LIN {X 0,Y 574.038,Z 321.65,A -85,B 0,C 180,E1 -2269.624,E2 -2269.624} C_VEL
LIN {X 0,Y 574.354,Z 297.27,A -85,B 0,C 180,E1 -2272.482,E2 -2272.482} C_VEL
LIN {X 0,Y 574.708,Z 273.214,A -85,B 0,C 180,E1 -2275.342,E2 -2275.342} C_VEL
LIN {X 0,Y 574.694,Z 268.348,A -85,B 0,C 180,E1 -2275.925,E2 -2275.925} C_VEL
LIN {X 0,Y 573.245,Z 261.708,A -85,B 0,C 180,E1 -2276.811,E2 -2276.811} C_VEL
LIN {X 0,Y 573.247,Z 261.7,A -85,B 0,C 180,E1 -2279.488,E2 -2279.488} C_VEL
LIN {X 0,Y 573.255,Z 261.706,A -85,B 0,C 180,E1 -2282.645,E2 -2282.645} C_VEL
LIN {X 0,Y 573.209,Z 261.705,A -85,B 0,C 180,E1 -2285.188,E2 -2285.188} C_VEL
LIN {X 0,Y 573.237,Z 261.701,A -85,B 0,C 180,E1 -2287.808,E2 -2287.808} C_VEL
LIN {X 0,Y 573.248,Z 261.707,A -85,B 0,C 180,E1 -2290.525,E2 -2290.525} C_VEL
LIN {X 0,Y 573.211,Z 261.703,A -85,B 0,C 180,E1 -2293.362,E2 -2293.362} C_VEL
LIN {X 0,Y 573.241,Z 261.707,A -85,B 0,C 180,E1 -2296.332,E2 -2296.332} C_VEL
LIN {X 0,Y 573.23,Z 261.707,A -85,B 0,C 180,E1 -2298.543,E2 -2298.543} C_VEL
LIN {X 0,Y 573.239,Z 261.699,A -85,B 0,C 180,E1 -2301.298,E2 -2301.298} C_VEL
LIN {X 0,Y 573.192,Z 261.711,A -85,B 0,C 180,E1 -2304.022,E2 -2304.022} C_VEL
LIN {X 0,Y 573.257,Z 261.702,A -85,B 0,C 180,E1 -2306.517,E2 -2306.517} C_VEL
LIN {X 0,Y 573.23,Z 261.7,A -85,B 0,C 180,E1 -2309.119,E2 -2309.119} C_VEL
LIN {X 0,Y 573.228,Z 261.7,A -85,B 0,C 180,E1 -2311.435,E2 -2311.435} C_VEL
LIN {X 0,Y 573.243,Z 261.702,A -85,B 0,C 180,E1 -2314.589,E2 -2314.589} C_VEL
LIN {X 0,Y 573.235,Z 261.702,A -85,B 0,C 180,E1 -2317.662,E2 -2317.662} C_VEL
LIN {X 0,Y 573.271,Z 261.696,A -85,B 0,C 180,E1 -2320.67,E2 -2320.67} C_VEL
LIN {X 0,Y 573.241,Z 261.703,A -85,B 0,C 180,E1 -2323.622,E2 -2323.622} C_VEL
LIN {X 0,Y 573.276,Z 261.7,A -85,B 0,C 180,E1 -2325.807,E2 -2325.807} C_VEL
LIN {X 0,Y 573.269,Z 261.695,A -85,B 0,C 180,E1 -2328.745,E2 -2328.745} C_VEL
LIN {X 0,Y 573.253,Z 261.701,A -85,B 0,C 180,E1 -2331.54,E2 -2331.54} C_VEL
LIN {X 0,Y 573.271,Z 261.698,A -85,B 0,C 180,E1 -2334.372,E2 -2334.372} C_VEL
LIN {X 0,Y 573.304,Z 261.7,A -85,B 0,C 180,E1 -2337.892,E2 -2337.892} C_VEL
LIN {X 0,Y 573.317,Z 261.697,A -85,B 0,C 180,E1 -2340,E2 -2340} C_VEL
LIN {X 0,Y 573.285,Z 261.693,A -85,B 0,C 180,E1 -2342.811,E2 -2342.811} C_VEL
LIN {X 0,Y 573.278,Z 261.702,A -85,B 0,C 180,E1 -2345.628,E2 -2345.628} C_VEL
LIN {X 0,Y 573.231,Z 261.701,A -85,B 0,C 180,E1 -2348.46,E2 -2348.46} C_VEL
LIN {X 0,Y 573.278,Z 261.697,A -85,B 0,C 180,E1 -2351.312,E2 -2351.312} C_VEL
LIN {X 0,Y 573.231,Z 261.7,A -85,B 0,C 180,E1 -2354.402,E2 -2354.402} C_VEL
LIN {X 0,Y 573.197,Z 261.707,A -85,B 0,C 180,E1 -2357.114,E2 -2357.114} C_VEL
LIN {X 0,Y 573.207,Z 261.706,A -85,B 0,C 180,E1 -2360.078,E2 -2360.078} C_VEL
LIN {X 0,Y 573.197,Z 261.704,A -85,B 0,C 180,E1 -2362.339,E2 -2362.339} C_VEL
LIN {X 0,Y 573.191,Z 261.706,A -85,B 0,C 180,E1 -2364.338,E2 -2364.338} C_VEL
LIN {X 0,Y 572.552,Z 261.787,A -85,B 0,C 180,E1 -2364.924,E2 -2364.924} C_VEL
LIN {X 0,Y 569.723,Z 262.146,A -85,B 0,C 180,E1 -2365.876,E2 -2365.876} C_VEL
LIN {X 0,Y 567.306,Z 262.45,A -85,B 0,C 180,E1 -2366.642,E2 -2366.642} C_VEL
LIN {X 0,Y 566.249,Z 262.577,A -85,B 0,C 180,E1 -2367.233,E2 -2367.233} C_VEL
LIN {X 0,Y 566.154,Z 262.586,A -85,B 0,C 180,E1 -2367.433,E2 -2367.433} C_VEL
LIN {X 0,Y 566.15,Z 262.587,A -85,B 0,C 180,E1 -2369.772,E2 -2369.772} C_VEL
LIN {X 0,Y 566.174,Z 262.579,A -85,B 0,C 180,E1 -2372.424,E2 -2372.424} C_VEL
LIN {X 0,Y 566.155,Z 262.585,A -85,B 0,C 180,E1 -2374.985,E2 -2374.985} C_VEL
LIN {X 0,Y 566.179,Z 262.587,A -85,B 0,C 180,E1 -2377.462,E2 -2377.462} C_VEL
LIN {X 0,Y 566.158,Z 262.581,A -85,B 0,C 180,E1 -2380.203,E2 -2380.203} C_VEL
LIN {X 0,Y 566.143,Z 262.589,A -85,B 0,C 180,E1 -2383.06,E2 -2383.06} C_VEL
LIN {X 0,Y 566.134,Z 262.584,A -85,B 0,C 180,E1 -2386.056,E2 -2386.056} C_VEL
LIN {X 0,Y 566.122,Z 262.589,A -85,B 0,C 180,E1 -2388.855,E2 -2388.855} C_VEL
LIN {X 0,Y 566.156,Z 262.587,A -85,B 0,C 180,E1 -2391.449,E2 -2391.449} C_VEL
LIN {X 0,Y 566.134,Z 262.585,A -85,B 0,C 180,E1 -2394.305,E2 -2394.305} C_VEL
LIN {X 0,Y 566.163,Z 262.586,A -85,B 0,C 180,E1 -2396.894,E2 -2396.894} C_VEL
LIN {X 0,Y 566.15,Z 262.588,A -85,B 0,C 180,E1 -2399.405,E2 -2399.405} C_VEL
LIN {X 0,Y 566.144,Z 262.585,A -85,B 0,C 180,E1 -2401.853,E2 -2401.853} C_VEL
LIN {X 0,Y 566.168,Z 262.582,A -85,B 0,C 180,E1 -2404.248,E2 -2404.248} C_VEL
LIN {X 0,Y 566.219,Z 262.756,A -85,B 0,C 180,E1 -2407.188,E2 -2407.188} C_VEL
LIN {X 0,Y 567.073,Z 267.816,A -85,B 0,C 180,E1 -2407.981,E2 -2407.981} C_VEL
LIN {X 0,Y 566.884,Z 283.111,A -85,B 0,C 180,E1 -2410.192,E2 -2410.192} C_VEL
LIN {X 0,Y 568.476,Z 291.01,A -85,B 0,C 180,E1 -2410.356,E2 -2410.356} C_VEL
LIN {X 0,Y 567.976,Z 448.126,A -85,B 0,C 180,E1 -2412.412,E2 -2412.412} C_VEL
LIN {X 0,Y 567.822,Z 463.751,A -85,B 0,C 180,E1 -2412.765,E2 -2412.765} C_VEL
LIN {X 0,Y 567.604,Z 479.067,A -85,B 0,C 180,E1 -2413.269,E2 -2413.269} C_VEL
LIN {X 0,Y 567.404,Z 493.725,A -85,B 0,C 180,E1 -2413.91,E2 -2413.91} C_VEL
LIN {X 0,Y 567.147,Z 507.039,A -85,B 0,C 180,E1 -2414.64,E2 -2414.64} C_VEL
LIN {X 0,Y 566.919,Z 519.973,A -85,B 0,C 180,E1 -2415.507,E2 -2415.507} C_VEL
LIN {X 0,Y 566.654,Z 532.884,A -85,B 0,C 180,E1 -2416.552,E2 -2416.552} C_VEL
LIN {X 0,Y 566.463,Z 544.081,A -85,B 0,C 180,E1 -2417.642,E2 -2417.642} C_VEL
LIN {X 0,Y 566.264,Z 554.176,A -85,B 0,C 180,E1 -2418.809,E2 -2418.809} C_VEL
LIN {X 0,Y 566.133,Z 564.001,A -85,B 0,C 180,E1 -2420.172,E2 -2420.172} C_VEL
LIN {X 0,Y 566.064,Z 571.492,A -85,B 0,C 180,E1 -2421.431,E2 -2421.431} C_VEL
LIN {X 0,Y 565.976,Z 578.497,A -85,B 0,C 180,E1 -2422.867,E2 -2422.867} C_VEL
LIN {X 0,Y 565.982,Z 584.007,A -85,B 0,C 180,E1 -2424.299,E2 -2424.299} C_VEL
LIN {X 0,Y 565.914,Z 588.177,A -85,B 0,C 180,E1 -2425.726,E2 -2425.726} C_VEL
LIN {X 0,Y 565.872,Z 591.113,A -85,B 0,C 180,E1 -2427.152,E2 -2427.152} C_VEL
LIN {X 0,Y 565.842,Z 592.879,A -85,B 0,C 180,E1 -2428.576,E2 -2428.576} C_VEL
LIN {X 0,Y 565.837,Z 593.496,A -85,B 0,C 180,E1 -2430,E2 -2430} C_VEL
LIN {X 0,Y 565.844,Z 592.941,A -85,B 0,C 180,E1 -2431.423,E2 -2431.423} C_VEL
LIN {X 0,Y 565.874,Z 591.258,A -85,B 0,C 180,E1 -2432.847,E2 -2432.847} C_VEL
LIN {X 0,Y 565.914,Z 588.404,A -85,B 0,C 180,E1 -2434.273,E2 -2434.273} C_VEL
LIN {X 0,Y 565.975,Z 584.319,A -85,B 0,C 180,E1 -2435.701,E2 -2435.701} C_VEL
LIN {X 0,Y 565.975,Z 578.905,A -85,B 0,C 180,E1 -2437.133,E2 -2437.133} C_VEL
LIN {X 0,Y 566.06,Z 572.004,A -85,B 0,C 180,E1 -2438.568,E2 -2438.568} C_VEL
LIN {X 0,Y 566.177,Z 563.396,A -85,B 0,C 180,E1 -2440.008,E2 -2440.008} C_VEL
LIN {X 0,Y 566.25,Z 554.953,A -85,B 0,C 180,E1 -2441.183,E2 -2441.183} C_VEL
LIN {X 0,Y 566.436,Z 544.917,A -85,B 0,C 180,E1 -2442.358,E2 -2442.358} C_VEL
LIN {X 0,Y 566.668,Z 532.874,A -85,B 0,C 180,E1 -2443.538,E2 -2443.538} C_VEL
LIN {X 0,Y 566.878,Z 521.25,A -85,B 0,C 180,E1 -2444.488,E2 -2444.488} C_VEL
LIN {X 0,Y 567.089,Z 508.476,A -85,B 0,C 180,E1 -2445.361,E2 -2445.361} C_VEL
LIN {X 0,Y 567.392,Z 495.466,A -85,B 0,C 180,E1 -2446.09,E2 -2446.09} C_VEL
LIN {X 0,Y 567.553,Z 481.274,A -85,B 0,C 180,E1 -2446.732,E2 -2446.732} C_VEL
LIN {X 0,Y 567.793,Z 466.726,A -85,B 0,C 180,E1 -2447.235,E2 -2447.235} C_VEL
LIN {X 0,Y 567.922,Z 451.446,A -85,B 0,C 180,E1 -2447.613,E2 -2447.613} C_VEL
LIN {X 0,Y 568.046,Z 429.928,A -85,B 0,C 180,E1 -2447.932,E2 -2447.932} C_VEL
LIN {X 0,Y 568.423,Z 290.393,A -85,B 0,C 180,E1 -2449.744,E2 -2449.744} C_VEL
LIN {X 0,Y 566.886,Z 283.074,A -85,B 0,C 180,E1 -2449.903,E2 -2449.903} C_VEL
LIN {X 0,Y 567.062,Z 267.137,A -85,B 0,C 180,E1 -2452.21,E2 -2452.21} C_VEL
LIN {X 0,Y 566.189,Z 262.587,A -85,B 0,C 180,E1 -2452.95,E2 -2452.95} C_VEL
LIN {X 0,Y 566.181,Z 262.581,A -85,B 0,C 180,E1 -2455.75,E2 -2455.75} C_VEL
LIN {X 0,Y 566.146,Z 262.585,A -85,B 0,C 180,E1 -2458.191,E2 -2458.191} C_VEL
LIN {X 0,Y 566.175,Z 262.589,A -85,B 0,C 180,E1 -2461.073,E2 -2461.073} C_VEL
LIN {X 0,Y 566.177,Z 262.581,A -85,B 0,C 180,E1 -2463.728,E2 -2463.728} C_VEL
LIN {X 0,Y 566.144,Z 262.588,A -85,B 0,C 180,E1 -2466.574,E2 -2466.574} C_VEL
LIN {X 0,Y 566.2,Z 262.58,A -85,B 0,C 180,E1 -2469.275,E2 -2469.275} C_VEL
LIN {X 0,Y 566.138,Z 262.585,A -85,B 0,C 180,E1 -2472.094,E2 -2472.094} C_VEL
LIN {X 0,Y 566.155,Z 262.588,A -85,B 0,C 180,E1 -2475.037,E2 -2475.037} C_VEL
LIN {X 0,Y 566.134,Z 262.583,A -85,B 0,C 180,E1 -2478.145,E2 -2478.145} C_VEL
LIN {X 0,Y 566.181,Z 262.589,A -85,B 0,C 180,E1 -2480.723,E2 -2480.723} C_VEL
LIN {X 0,Y 566.136,Z 262.58,A -85,B 0,C 180,E1 -2483.425,E2 -2483.425} C_VEL
LIN {X 0,Y 566.174,Z 262.583,A -85,B 0,C 180,E1 -2486.271,E2 -2486.271} C_VEL
LIN {X 0,Y 566.167,Z 262.585,A -85,B 0,C 180,E1 -2488.927,E2 -2488.927} C_VEL
LIN {X 0,Y 566.138,Z 262.584,A -85,B 0,C 180,E1 -2491.853,E2 -2491.853} C_VEL
LIN {X 0,Y 566.173,Z 262.584,A -85,B 0,C 180,E1 -2494.249,E2 -2494.249} C_VEL
LIN {X 0,Y 566.145,Z 262.589,A -85,B 0,C 180,E1 -2496.725,E2 -2496.725} C_VEL
LIN {X 0,Y 566.181,Z 262.582,A -85,B 0,C 180,E1 -2498.901,E2 -2498.901} C_VEL
LIN {X 0,Y 566.181,Z 262.578,A -85,B 0,C 180,E1 -2501.171,E2 -2501.171} C_VEL
LIN {X 0,Y 566.167,Z 262.586,A -85,B 0,C 180,E1 -2504.152,E2 -2504.152} C_VEL
LIN {X 0,Y 566.156,Z 262.59,A -85,B 0,C 180,E1 -2506.358,E2 -2506.358} C_VEL
LIN {X 0,Y 566.217,Z 262.574,A -85,B 0,C 180,E1 -2509.27,E2 -2509.27} C_VEL
LIN {X 0,Y 566.199,Z 262.582,A -85,B 0,C 180,E1 -2512.152,E2 -2512.152} C_VEL
LIN {X 0,Y 566.254,Z 262.569,A -85,B 0,C 180,E1 -2515.016,E2 -2515.016} C_VEL
LIN {X 0,Y 566.267,Z 262.571,A -85,B 0,C 180,E1 -2517.866,E2 -2517.866} C_VEL
LIN {X 0,Y 566.295,Z 262.565,A -85,B 0,C 180,E1 -2520.711,E2 -2520.711} C_VEL
LIN {X 0,Y 566.255,Z 262.57,A -85,B 0,C 180,E1 -2522.846,E2 -2522.846} C_VEL
LIN {X 0,Y 566.236,Z 262.574,A -85,B 0,C 180,E1 -2525.698,E2 -2525.698} C_VEL
LIN {X 0,Y 566.199,Z 262.579,A -85,B 0,C 180,E1 -2528.566,E2 -2528.566} C_VEL
LIN {X 0,Y 566.241,Z 262.571,A -85,B 0,C 180,E1 -2531.454,E2 -2531.454} C_VEL
LIN {X 0,Y 566.233,Z 262.574,A -85,B 0,C 180,E1 -2534.506,E2 -2534.506} C_VEL
LIN {X 0,Y 566.192,Z 262.579,A -85,B 0,C 180,E1 -2537.332,E2 -2537.332} C_VEL
LIN {X 0,Y 566.204,Z 262.58,A -85,B 0,C 180,E1 -2540.337,E2 -2540.337} C_VEL
LIN {X 0,Y 566.167,Z 262.581,A -85,B 0,C 180,E1 -2543.28,E2 -2543.28} C_VEL
LIN {X 0,Y 566.206,Z 262.579,A -85,B 0,C 180,E1 -2545.749,E2 -2545.749} C_VEL
LIN {X 0,Y 566.183,Z 262.579,A -85,B 0,C 180,E1 -2548.954,E2 -2548.954} C_VEL
LIN {X 0,Y 566.191,Z 262.58,A -85,B 0,C 180,E1 -2551.422,E2 -2551.422} C_VEL
LIN {X 0,Y 566.207,Z 262.582,A -85,B 0,C 180,E1 -2553.956,E2 -2553.956} C_VEL
LIN {X 0,Y 566.206,Z 262.574,A -85,B 0,C 180,E1 -2556.569,E2 -2556.569} C_VEL
LIN {X 0,Y 566.212,Z 262.584,A -85,B 0,C 180,E1 -2559.686,E2 -2559.686} C_VEL
LIN {X 0,Y 566.199,Z 262.577,A -85,B 0,C 180,E1 -2562.917,E2 -2562.917} C_VEL
LIN {X 0,Y 566.192,Z 262.58,A -85,B 0,C 180,E1 -2566.049,E2 -2566.049} C_VEL
LIN {X 0,Y 566.174,Z 262.58,A -85,B 0,C 180,E1 -2568.861,E2 -2568.861} C_VEL
LIN {X 0,Y 566.209,Z 262.584,A -85,B 0,C 180,E1 -2571.442,E2 -2571.442} C_VEL
LIN {X 0,Y 566.195,Z 262.578,A -85,B 0,C 180,E1 -2574.311,E2 -2574.311} C_VEL
LIN {X 0,Y 566.219,Z 262.576,A -85,B 0,C 180,E1 -2576.898,E2 -2576.898} C_VEL
LIN {X 0,Y 566.18,Z 262.588,A -85,B 0,C 180,E1 -2579.407,E2 -2579.407} C_VEL
LIN {X 0,Y 566.211,Z 262.582,A -85,B 0,C 180,E1 -2581.858,E2 -2581.858} C_VEL
LIN {X 0,Y 566.242,Z 262.647,A -85,B 0,C 180,E1 -2582.997,E2 -2582.997} C_VEL
LIN {X 0,Y 567.807,Z 269.73,A -85,B 0,C 180,E1 -2583.935,E2 -2583.935} C_VEL
LIN {X 0,Y 567.648,Z 288.822,A -85,B 0,C 180,E1 -2586.231,E2 -2586.231} C_VEL
LIN {X 0,Y 567.281,Z 313.234,A -85,B 0,C 180,E1 -2589.134,E2 -2589.134} C_VEL
LIN {X 0,Y 567.133,Z 321.683,A -85,B 0,C 180,E1 -2590.131,E2 -2590.131} C_VEL
LIN {X 0,Y 568.538,Z 330.177,A -85,B 0,C 180,E1 -2590.303,E2 -2590.303} C_VEL
LIN {X 0,Y 567.993,Z 488.227,A -85,B 0,C 180,E1 -2592.369,E2 -2592.369} C_VEL
LIN {X 0,Y 567.834,Z 503.714,A -85,B 0,C 180,E1 -2592.72,E2 -2592.72} C_VEL
LIN {X 0,Y 567.61,Z 519.045,A -85,B 0,C 180,E1 -2593.223,E2 -2593.223} C_VEL
LIN {X 0,Y 567.445,Z 532.78,A -85,B 0,C 180,E1 -2593.819,E2 -2593.819} C_VEL
LIN {X 0,Y 567.151,Z 546.252,A -85,B 0,C 180,E1 -2594.549,E2 -2594.549} C_VEL
LIN {X 0,Y 566.922,Z 559.506,A -85,B 0,C 180,E1 -2595.429,E2 -2595.429} C_VEL
LIN {X 0,Y 566.674,Z 572.355,A -85,B 0,C 180,E1 -2596.462,E2 -2596.462} C_VEL
LIN {X 0,Y 566.491,Z 582.752,A -85,B 0,C 180,E1 -2597.461,E2 -2597.461} C_VEL
LIN {X 0,Y 566.268,Z 593.314,A -85,B 0,C 180,E1 -2598.659,E2 -2598.659} C_VEL
LIN {X 0,Y 566.208,Z 601.859,A -85,B 0,C 180,E1 -2599.812,E2 -2599.812} C_VEL
LIN {X 0,Y 566.057,Z 609.736,A -85,B 0,C 180,E1 -2601.072,E2 -2601.072} C_VEL
LIN {X 0,Y 565.997,Z 617.091,A -85,B 0,C 180,E1 -2602.509,E2 -2602.509} C_VEL
LIN {X 0,Y 565.956,Z 622.924,A -85,B 0,C 180,E1 -2603.941,E2 -2603.941} C_VEL
LIN {X 0,Y 565.866,Z 626.387,A -85,B 0,C 180,E1 -2605.013,E2 -2605.013} C_VEL
LIN {X 0,Y 565.909,Z 629.89,A -85,B 0,C 180,E1 -2606.44,E2 -2606.44} C_VEL
LIN {X 0,Y 565.838,Z 632.192,A -85,B 0,C 180,E1 -2607.865,E2 -2607.865} C_VEL
LIN {X 0,Y 565.838,Z 633.349,A -85,B 0,C 180,E1 -2609.289,E2 -2609.289} C_VEL
LIN {X 0,Y 565.838,Z 633.348,A -85,B 0,C 180,E1 -2610.712,E2 -2610.712} C_VEL
LIN {X 0,Y 565.838,Z 632.189,A -85,B 0,C 180,E1 -2612.136,E2 -2612.136} C_VEL
LIN {X 0,Y 565.909,Z 629.886,A -85,B 0,C 180,E1 -2613.56,E2 -2613.56} C_VEL
LIN {X 0,Y 565.866,Z 626.385,A -85,B 0,C 180,E1 -2614.988,E2 -2614.988} C_VEL
LIN {X 0,Y 565.956,Z 622.923,A -85,B 0,C 180,E1 -2616.059,E2 -2616.059} C_VEL
LIN {X 0,Y 565.998,Z 617.086,A -85,B 0,C 180,E1 -2617.492,E2 -2617.492} C_VEL
LIN {X 0,Y 566.058,Z 609.729,A -85,B 0,C 180,E1 -2618.929,E2 -2618.929} C_VEL
LIN {X 0,Y 566.208,Z 601.853,A -85,B 0,C 180,E1 -2620.188,E2 -2620.188} C_VEL
LIN {X 0,Y 566.309,Z 592.387,A -85,B 0,C 180,E1 -2621.453,E2 -2621.453} C_VEL
LIN {X 0,Y 566.492,Z 582.745,A -85,B 0,C 180,E1 -2622.54,E2 -2622.54} C_VEL
LIN {X 0,Y 566.672,Z 571.29,A -85,B 0,C 180,E1 -2623.63,E2 -2623.63} C_VEL
LIN {X 0,Y 566.95,Z 558.671,A -85,B 0,C 180,E1 -2624.63,E2 -2624.63} C_VEL
LIN {X 0,Y 567.148,Z 546.239,A -85,B 0,C 180,E1 -2625.452,E2 -2625.452} C_VEL
LIN {X 0,Y 567.448,Z 532.759,A -85,B 0,C 180,E1 -2626.181,E2 -2626.181} C_VEL
LIN {X 0,Y 567.612,Z 519.035,A -85,B 0,C 180,E1 -2626.777,E2 -2626.777} C_VEL
LIN {X 0,Y 567.849,Z 503.702,A -85,B 0,C 180,E1 -2627.28,E2 -2627.28} C_VEL
LIN {X 0,Y 567.982,Z 488.271,A -85,B 0,C 180,E1 -2627.63,E2 -2627.63} C_VEL
LIN {X 0,Y 568.52,Z 329.185,A -85,B 0,C 180,E1 -2629.711,E2 -2629.711} C_VEL
LIN {X 0,Y 567.141,Z 321.689,A -85,B 0,C 180,E1 -2629.868,E2 -2629.868} C_VEL
LIN {X 0,Y 567.533,Z 297.268,A -85,B 0,C 180,E1 -2632.767,E2 -2632.767} C_VEL
LIN {X 0,Y 567.908,Z 271.347,A -85,B 0,C 180,E1 -2635.864,E2 -2635.864} C_VEL
LIN {X 0,Y 567.091,Z 266.447,A -85,B 0,C 180,E1 -2636.497,E2 -2636.497} C_VEL
LIN {X 0,Y 566.229,Z 262.581,A -85,B 0,C 180,E1 -2637.026,E2 -2637.026} C_VEL
LIN {X 0,Y 566.202,Z 262.578,A -85,B 0,C 180,E1 -2639.769,E2 -2639.769} C_VEL
LIN {X 0,Y 566.206,Z 262.584,A -85,B 0,C 180,E1 -2642.43,E2 -2642.43} C_VEL
LIN {X 0,Y 566.182,Z 262.582,A -85,B 0,C 180,E1 -2644.99,E2 -2644.99} C_VEL
LIN {X 0,Y 566.198,Z 262.576,A -85,B 0,C 180,E1 -2647.461,E2 -2647.461} C_VEL
LIN {X 0,Y 566.21,Z 262.579,A -85,B 0,C 180,E1 -2650.199,E2 -2650.199} C_VEL
LIN {X 0,Y 566.19,Z 262.579,A -85,B 0,C 180,E1 -2653.056,E2 -2653.056} C_VEL
LIN {X 0,Y 566.197,Z 262.581,A -85,B 0,C 180,E1 -2656.05,E2 -2656.05} C_VEL
LIN {X 0,Y 566.207,Z 262.575,A -85,B 0,C 180,E1 -2659.215,E2 -2659.215} C_VEL
LIN {X 0,Y 566.185,Z 262.579,A -85,B 0,C 180,E1 -2661.637,E2 -2661.637} C_VEL
LIN {X 0,Y 566.148,Z 262.591,A -85,B 0,C 180,E1 -2664.307,E2 -2664.307} C_VEL
LIN {X 0,Y 566.215,Z 262.575,A -85,B 0,C 180,E1 -2666.898,E2 -2666.898} C_VEL
LIN {X 0,Y 566.182,Z 262.578,A -85,B 0,C 180,E1 -2669.407,E2 -2669.407} C_VEL
LIN {X 0,Y 566.191,Z 262.581,A -85,B 0,C 180,E1 -2671.856,E2 -2671.856} C_VEL
LIN {X 0,Y 566.242,Z 262.571,A -85,B 0,C 180,E1 -2675.039,E2 -2675.039} C_VEL
LIN {X 0,Y 566.196,Z 262.586,A -85,B 0,C 180,E1 -2678.138,E2 -2678.138} C_VEL
LIN {X 0,Y 566.236,Z 262.573,A -85,B 0,C 180,E1 -2680.614,E2 -2680.614} C_VEL
LIN {X 0,Y 566.204,Z 262.577,A -85,B 0,C 180,E1 -2683.412,E2 -2683.412} C_VEL
LIN {X 0,Y 566.192,Z 262.582,A -85,B 0,C 180,E1 -2686.359,E2 -2686.359} C_VEL
LIN {X 0,Y 566.241,Z 262.571,A -85,B 0,C 180,E1 -2688.676,E2 -2688.676} C_VEL
LIN {X 0,Y 566.204,Z 262.578,A -85,B 0,C 180,E1 -2691.434,E2 -2691.434} C_VEL
LIN {X 0,Y 566.241,Z 262.575,A -85,B 0,C 180,E1 -2694.302,E2 -2694.302} C_VEL
LIN {X 0,Y 566.276,Z 262.575,A -85,B 0,C 180,E1 -2697.866,E2 -2697.866} C_VEL
LIN {X 0,Y 566.286,Z 262.572,A -85,B 0,C 180,E1 -2700,E2 -2700} C_VEL
LIN {X 0,Y 566.254,Z 262.569,A -85,B 0,C 180,E1 -2702.846,E2 -2702.846} C_VEL
LIN {X 0,Y 566.244,Z 262.579,A -85,B 0,C 180,E1 -2705.699,E2 -2705.699} C_VEL
LIN {X 0,Y 566.185,Z 262.578,A -85,B 0,C 180,E1 -2708.566,E2 -2708.566} C_VEL
LIN {X 0,Y 566.244,Z 262.575,A -85,B 0,C 180,E1 -2711.454,E2 -2711.454} C_VEL
LIN {X 0,Y 566.181,Z 262.577,A -85,B 0,C 180,E1 -2714.483,E2 -2714.483} C_VEL
LIN {X 0,Y 566.162,Z 262.586,A -85,B 0,C 180,E1 -2717.333,E2 -2717.333} C_VEL
LIN {X 0,Y 566.178,Z 262.587,A -85,B 0,C 180,E1 -2719.582,E2 -2719.582} C_VEL
LIN {X 0,Y 566.15,Z 262.587,A -85,B 0,C 180,E1 -2721.864,E2 -2721.864} C_VEL
LIN {X 0,Y 566.145,Z 262.584,A -85,B 0,C 180,E1 -2724.335,E2 -2724.335} C_VEL
LIN {X 0,Y 566.174,Z 262.578,A -85,B 0,C 180,E1 -2726.651,E2 -2726.651} C_VEL
LIN {X 0,Y 566.154,Z 262.586,A -85,B 0,C 180,E1 -2727.433,E2 -2727.433} C_VEL
LIN {X 0,Y 565.458,Z 262.668,A -85,B 0,C 180,E1 -2728.027,E2 -2728.027} C_VEL
LIN {X 0,Y 562.584,Z 263.025,A -85,B 0,C 180,E1 -2728.991,E2 -2728.991} C_VEL
LIN {X 0,Y 560.184,Z 263.331,A -85,B 0,C 180,E1 -2729.766,E2 -2729.766} C_VEL
LIN {X 0,Y 559.173,Z 263.452,A -85,B 0,C 180,E1 -2730.365,E2 -2730.365} C_VEL
LIN {X 0,Y 559.1,Z 263.46,A -85,B 0,C 180,E1 -2730.568,E2 -2730.568} C_VEL
LIN {X 0,Y 559.136,Z 263.457,A -85,B 0,C 180,E1 -2732.717,E2 -2732.717} C_VEL
LIN {X 0,Y 559.112,Z 263.468,A -85,B 0,C 180,E1 -2735.325,E2 -2735.325} C_VEL
LIN {X 0,Y 559.099,Z 263.461,A -85,B 0,C 180,E1 -2738.02,E2 -2738.02} C_VEL
LIN {X 0,Y 559.093,Z 263.464,A -85,B 0,C 180,E1 -2740.818,E2 -2740.818} C_VEL
LIN {X 0,Y 559.093,Z 263.464,A -85,B 0,C 180,E1 -2743.739,E2 -2743.739} C_VEL
LIN {X 0,Y 559.084,Z 263.462,A -85,B 0,C 180,E1 -2746.26,E2 -2746.26} C_VEL
LIN {X 0,Y 559.085,Z 263.471,A -85,B 0,C 180,E1 -2749.181,E2 -2749.181} C_VEL
LIN {X 0,Y 559.115,Z 263.469,A -85,B 0,C 180,E1 -2751.2,E2 -2751.2} C_VEL
LIN {X 0,Y 559.11,Z 263.462,A -85,B 0,C 180,E1 -2753.786,E2 -2753.786} C_VEL
LIN {X 0,Y 559.115,Z 263.459,A -85,B 0,C 180,E1 -2756.421,E2 -2756.421} C_VEL
LIN {X 0,Y 559.136,Z 263.463,A -85,B 0,C 180,E1 -2758.979,E2 -2758.979} C_VEL
LIN {X 0,Y 559.105,Z 263.463,A -85,B 0,C 180,E1 -2761.631,E2 -2761.631} C_VEL
LIN {X 0,Y 559.116,Z 263.461,A -85,B 0,C 180,E1 -2763.899,E2 -2763.899} C_VEL
LIN {X 0,Y 559.16,Z 263.488,A -85,B 0,C 180,E1 -2766.96,E2 -2766.96} C_VEL
LIN {X 0,Y 560.198,Z 269.356,A -85,B 0,C 180,E1 -2767.891,E2 -2767.891} C_VEL
LIN {X 0,Y 560.006,Z 283.147,A -85,B 0,C 180,E1 -2769.939,E2 -2769.939} C_VEL
LIN {X 0,Y 561.793,Z 292.249,A -85,B 0,C 180,E1 -2770.129,E2 -2770.129} C_VEL
LIN {X 0,Y 561.22,Z 448.397,A -85,B 0,C 180,E1 -2772.198,E2 -2772.198} C_VEL
LIN {X 0,Y 561.06,Z 463.772,A -85,B 0,C 180,E1 -2772.551,E2 -2772.551} C_VEL
LIN {X 0,Y 560.795,Z 479.08,A -85,B 0,C 180,E1 -2773.059,E2 -2773.059} C_VEL
LIN {X 0,Y 560.572,Z 493.733,A -85,B 0,C 180,E1 -2773.708,E2 -2773.708} C_VEL
LIN {X 0,Y 560.244,Z 507.051,A -85,B 0,C 180,E1 -2774.446,E2 -2774.446} C_VEL
LIN {X 0,Y 559.985,Z 520.385,A -85,B 0,C 180,E1 -2775.353,E2 -2775.353} C_VEL
LIN {X 0,Y 559.691,Z 532.892,A -85,B 0,C 180,E1 -2776.382,E2 -2776.382} C_VEL
LIN {X 0,Y 559.487,Z 544.087,A -85,B 0,C 180,E1 -2777.485,E2 -2777.485} C_VEL
LIN {X 0,Y 559.229,Z 554.785,A -85,B 0,C 180,E1 -2778.743,E2 -2778.743} C_VEL
LIN {X 0,Y 559.096,Z 564.004,A -85,B 0,C 180,E1 -2780.047,E2 -2780.047} C_VEL
LIN {X 0,Y 559.003,Z 571.495,A -85,B 0,C 180,E1 -2781.322,E2 -2781.322} C_VEL
LIN {X 0,Y 558.901,Z 578.5,A -85,B 0,C 180,E1 -2782.776,E2 -2782.776} C_VEL
LIN {X 0,Y 558.887,Z 584.01,A -85,B 0,C 180,E1 -2784.226,E2 -2784.226} C_VEL
LIN {X 0,Y 558.809,Z 588.178,A -85,B 0,C 180,E1 -2785.672,E2 -2785.672} C_VEL
LIN {X 0,Y 558.793,Z 591.112,A -85,B 0,C 180,E1 -2787.116,E2 -2787.116} C_VEL
LIN {X 0,Y 558.742,Z 592.879,A -85,B 0,C 180,E1 -2788.558,E2 -2788.558} C_VEL
LIN {X 0,Y 558.738,Z 593.496,A -85,B 0,C 180,E1 -2790,E2 -2790} C_VEL
LIN {X 0,Y 558.744,Z 592.94,A -85,B 0,C 180,E1 -2791.441,E2 -2791.441} C_VEL
LIN {X 0,Y 558.795,Z 591.256,A -85,B 0,C 180,E1 -2792.883,E2 -2792.883} C_VEL
LIN {X 0,Y 558.809,Z 588.403,A -85,B 0,C 180,E1 -2794.327,E2 -2794.327} C_VEL
LIN {X 0,Y 558.88,Z 584.317,A -85,B 0,C 180,E1 -2795.773,E2 -2795.773} C_VEL
LIN {X 0,Y 558.9,Z 578.902,A -85,B 0,C 180,E1 -2797.224,E2 -2797.224} C_VEL
LIN {X 0,Y 559,Z 572.001,A -85,B 0,C 180,E1 -2798.677,E2 -2798.677} C_VEL
LIN {X 0,Y 559.091,Z 564.573,A -85,B 0,C 180,E1 -2799.953,E2 -2799.953} C_VEL
LIN {X 0,Y 559.215,Z 555.512,A -85,B 0,C 180,E1 -2801.25,E2 -2801.25} C_VEL
LIN {X 0,Y 559.451,Z 544.911,A -85,B 0,C 180,E1 -2802.515,E2 -2802.515} C_VEL
LIN {X 0,Y 559.696,Z 532.867,A -85,B 0,C 180,E1 -2803.71,E2 -2803.71} C_VEL
LIN {X 0,Y 559.998,Z 520.175,A -85,B 0,C 180,E1 -2804.751,E2 -2804.751} C_VEL
LIN {X 0,Y 560.272,Z 507.01,A -85,B 0,C 180,E1 -2805.646,E2 -2805.646} C_VEL
LIN {X 0,Y 560.568,Z 493.686,A -85,B 0,C 180,E1 -2806.385,E2 -2806.385} C_VEL
LIN {X 0,Y 560.813,Z 478.995,A -85,B 0,C 180,E1 -2807.033,E2 -2807.033} C_VEL
LIN {X 0,Y 561.079,Z 463.519,A -85,B 0,C 180,E1 -2807.545,E2 -2807.545} C_VEL
LIN {X 0,Y 561.216,Z 447.602,A -85,B 0,C 180,E1 -2807.907,E2 -2807.907} C_VEL
LIN {X 0,Y 561.818,Z 292.16,A -85,B 0,C 180,E1 -2809.962,E2 -2809.962} C_VEL
LIN {X 0,Y 559.989,Z 282.991,A -85,B 0,C 180,E1 -2810.175,E2 -2810.175} C_VEL
LIN {X 0,Y 560.184,Z 268.67,A -85,B 0,C 180,E1 -2812.303,E2 -2812.303} C_VEL
LIN {X 0,Y 559.131,Z 263.467,A -85,B 0,C 180,E1 -2813.149,E2 -2813.149} C_VEL
LIN {X 0,Y 559.147,Z 263.456,A -85,B 0,C 180,E1 -2816.098,E2 -2816.098} C_VEL
LIN {X 0,Y 559.105,Z 263.465,A -85,B 0,C 180,E1 -2818.533,E2 -2818.533} C_VEL
LIN {X 0,Y 559.122,Z 263.465,A -85,B 0,C 180,E1 -2821.269,E2 -2821.269} C_VEL
LIN {X 0,Y 559.138,Z 263.458,A -85,B 0,C 180,E1 -2823.945,E2 -2823.945} C_VEL
LIN {X 0,Y 559.112,Z 263.467,A -85,B 0,C 180,E1 -2827.11,E2 -2827.11} C_VEL
LIN {X 0,Y 559.152,Z 263.455,A -85,B 0,C 180,E1 -2829.94,E2 -2829.94} C_VEL
LIN {X 0,Y 559.093,Z 263.464,A -85,B 0,C 180,E1 -2833.19,E2 -2833.19} C_VEL
LIN {X 0,Y 559.112,Z 263.459,A -85,B 0,C 180,E1 -2835.765,E2 -2835.765} C_VEL
LIN {X 0,Y 559.091,Z 263.46,A -85,B 0,C 180,E1 -2838.223,E2 -2838.223} C_VEL
LIN {X 0,Y 559.12,Z 263.462,A -85,B 0,C 180,E1 -2841.061,E2 -2841.061} C_VEL
LIN {X 0,Y 559.104,Z 263.455,A -85,B 0,C 180,E1 -2843.786,E2 -2843.786} C_VEL
LIN {X 0,Y 559.12,Z 263.464,A -85,B 0,C 180,E1 -2846.422,E2 -2846.422} C_VEL
LIN {X 0,Y 559.132,Z 263.46,A -85,B 0,C 180,E1 -2848.979,E2 -2848.979} C_VEL
LIN {X 0,Y 559.1,Z 263.46,A -85,B 0,C 180,E1 -2851.632,E2 -2851.632} C_VEL
LIN {X 0,Y 559.12,Z 263.465,A -85,B 0,C 180,E1 -2854.699,E2 -2854.699} C_VEL
LIN {X 0,Y 559.089,Z 263.463,A -85,B 0,C 180,E1 -2857.065,E2 -2857.065} C_VEL
LIN {X 0,Y 559.11,Z 263.459,A -85,B 0,C 180,E1 -2859.393,E2 -2859.393} C_VEL
LIN {X 0,Y 559.112,Z 263.458,A -85,B 0,C 180,E1 -2861.684,E2 -2861.684} C_VEL
LIN {X 0,Y 559.125,Z 263.461,A -85,B 0,C 180,E1 -2864.695,E2 -2864.695} C_VEL
LIN {X 0,Y 559.139,Z 263.456,A -85,B 0,C 180,E1 -2867.662,E2 -2867.662} C_VEL
LIN {X 0,Y 559.115,Z 263.461,A -85,B 0,C 180,E1 -2869.864,E2 -2869.864} C_VEL
LIN {X 0,Y 559.174,Z 263.455,A -85,B 0,C 180,E1 -2872.053,E2 -2872.053} C_VEL
LIN {X 0,Y 559.23,Z 263.444,A -85,B 0,C 180,E1 -2874.953,E2 -2874.953} C_VEL
LIN {X 0,Y 559.239,Z 263.447,A -85,B 0,C 180,E1 -2877.839,E2 -2877.839} C_VEL
LIN {X 0,Y 559.266,Z 263.44,A -85,B 0,C 180,E1 -2880.72,E2 -2880.72} C_VEL
LIN {X 0,Y 559.221,Z 263.446,A -85,B 0,C 180,E1 -2882.881,E2 -2882.881} C_VEL
LIN {X 0,Y 559.207,Z 263.451,A -85,B 0,C 180,E1 -2885.77,E2 -2885.77} C_VEL
LIN {X 0,Y 559.163,Z 263.454,A -85,B 0,C 180,E1 -2888.675,E2 -2888.675} C_VEL
LIN {X 0,Y 559.203,Z 263.449,A -85,B 0,C 180,E1 -2891.6,E2 -2891.6} C_VEL
LIN {X 0,Y 559.2,Z 263.449,A -85,B 0,C 180,E1 -2894.595,E2 -2894.595} C_VEL
LIN {X 0,Y 559.135,Z 263.46,A -85,B 0,C 180,E1 -2897.558,E2 -2897.558} C_VEL
LIN {X 0,Y 559.164,Z 263.46,A -85,B 0,C 180,E1 -2899.838,E2 -2899.838} C_VEL
LIN {X 0,Y 559.138,Z 263.461,A -85,B 0,C 180,E1 -2902.153,E2 -2902.153} C_VEL
LIN {X 0,Y 559.174,Z 263.448,A -85,B 0,C 180,E1 -2905.298,E2 -2905.298} C_VEL
LIN {X 0,Y 559.125,Z 263.464,A -85,B 0,C 180,E1 -2907.715,E2 -2907.715} C_VEL
LIN {X 0,Y 559.15,Z 263.456,A -85,B 0,C 180,E1 -2910.183,E2 -2910.183} C_VEL
LIN {X 0,Y 559.155,Z 263.451,A -85,B 0,C 180,E1 -2912.715,E2 -2912.715} C_VEL
LIN {X 0,Y 559.141,Z 263.459,A -85,B 0,C 180,E1 -2915.323,E2 -2915.323} C_VEL
LIN {X 0,Y 559.13,Z 263.461,A -85,B 0,C 180,E1 -2918.018,E2 -2918.018} C_VEL
LIN {X 0,Y 559.154,Z 263.454,A -85,B 0,C 180,E1 -2920.813,E2 -2920.813} C_VEL
LIN {X 0,Y 559.136,Z 263.465,A -85,B 0,C 180,E1 -2923.734,E2 -2923.734} C_VEL
LIN {X 0,Y 559.143,Z 263.455,A -85,B 0,C 180,E1 -2926.804,E2 -2926.804} C_VEL
LIN {X 0,Y 559.155,Z 263.457,A -85,B 0,C 180,E1 -2929.188,E2 -2929.188} C_VEL
LIN {X 0,Y 559.132,Z 263.46,A -85,B 0,C 180,E1 -2931.983,E2 -2931.983} C_VEL
LIN {X 0,Y 559.146,Z 263.457,A -85,B 0,C 180,E1 -2934.785,E2 -2934.785} C_VEL
LIN {X 0,Y 559.155,Z 263.463,A -85,B 0,C 180,E1 -2937.365,E2 -2937.365} C_VEL
LIN {X 0,Y 559.148,Z 263.458,A -85,B 0,C 180,E1 -2940.143,E2 -2940.143} C_VEL
LIN {X 0,Y 559.209,Z 263.586,A -85,B 0,C 180,E1 -2942.779,E2 -2942.779} C_VEL
LIN {X 0,Y 561.076,Z 272.724,A -85,B 0,C 180,E1 -2943.998,E2 -2943.998} C_VEL
LIN {X 0,Y 560.65,Z 298.635,A -85,B 0,C 180,E1 -2947.133,E2 -2947.133} C_VEL
LIN {X 0,Y 560.304,Z 322.054,A -85,B 0,C 180,E1 -2949.892,E2 -2949.892} C_VEL
LIN {X 0,Y 561.873,Z 330.795,A -85,B 0,C 180,E1 -2950.067,E2 -2950.067} C_VEL
LIN {X 0,Y 561.242,Z 488.226,A -85,B 0,C 180,E1 -2952.15,E2 -2952.15} C_VEL
LIN {X 0,Y 561.061,Z 503.713,A -85,B 0,C 180,E1 -2952.505,E2 -2952.505} C_VEL
LIN {X 0,Y 560.813,Z 519.043,A -85,B 0,C 180,E1 -2953.014,E2 -2953.014} C_VEL
LIN {X 0,Y 560.606,Z 532.783,A -85,B 0,C 180,E1 -2953.617,E2 -2953.617} C_VEL
LIN {X 0,Y 560.286,Z 546.255,A -85,B 0,C 180,E1 -2954.355,E2 -2954.355} C_VEL
LIN {X 0,Y 560,Z 559.29,A -85,B 0,C 180,E1 -2955.229,E2 -2955.229} C_VEL
LIN {X 0,Y 559.722,Z 571.296,A -85,B 0,C 180,E1 -2956.198,E2 -2956.198} C_VEL
LIN {X 0,Y 559.516,Z 582.752,A -85,B 0,C 180,E1 -2957.302,E2 -2957.302} C_VEL
LIN {X 0,Y 559.303,Z 592.392,A -85,B 0,C 180,E1 -2958.402,E2 -2958.402} C_VEL
LIN {X 0,Y 559.168,Z 601.858,A -85,B 0,C 180,E1 -2959.683,E2 -2959.683} C_VEL
LIN {X 0,Y 559.003,Z 609.737,A -85,B 0,C 180,E1 -2960.959,E2 -2960.959} C_VEL
LIN {X 0,Y 558.92,Z 617.091,A -85,B 0,C 180,E1 -2962.413,E2 -2962.413} C_VEL
LIN {X 0,Y 558.858,Z 622.923,A -85,B 0,C 180,E1 -2963.864,E2 -2963.864} C_VEL
LIN {X 0,Y 558.787,Z 626.387,A -85,B 0,C 180,E1 -2964.949,E2 -2964.949} C_VEL
LIN {X 0,Y 558.818,Z 629.89,A -85,B 0,C 180,E1 -2966.395,E2 -2966.395} C_VEL
LIN {X 0,Y 558.744,Z 632.191,A -85,B 0,C 180,E1 -2967.838,E2 -2967.838} C_VEL
LIN {X 0,Y 558.739,Z 633.349,A -85,B 0,C 180,E1 -2969.28,E2 -2969.28} C_VEL
LIN {X 0,Y 558.739,Z 633.348,A -85,B 0,C 180,E1 -2970.721,E2 -2970.721} C_VEL
LIN {X 0,Y 558.744,Z 632.188,A -85,B 0,C 180,E1 -2972.163,E2 -2972.163} C_VEL
LIN {X 0,Y 558.818,Z 629.885,A -85,B 0,C 180,E1 -2973.606,E2 -2973.606} C_VEL
LIN {X 0,Y 558.787,Z 626.385,A -85,B 0,C 180,E1 -2975.051,E2 -2975.051} C_VEL
LIN {X 0,Y 558.843,Z 621.607,A -85,B 0,C 180,E1 -2976.499,E2 -2976.499} C_VEL
LIN {X 0,Y 558.951,Z 615.42,A -85,B 0,C 180,E1 -2977.95,E2 -2977.95} C_VEL
LIN {X 0,Y 559.005,Z 607.643,A -85,B 0,C 180,E1 -2979.407,E2 -2979.407} C_VEL
LIN {X 0,Y 559.217,Z 599.365,A -85,B 0,C 180,E1 -2980.683,E2 -2980.683} C_VEL
LIN {X 0,Y 559.363,Z 589.388,A -85,B 0,C 180,E1 -2981.965,E2 -2981.965} C_VEL
LIN {X 0,Y 559.597,Z 579.182,A -85,B 0,C 180,E1 -2983.066,E2 -2983.066} C_VEL
LIN {X 0,Y 559.825,Z 567.014,A -85,B 0,C 180,E1 -2984.17,E2 -2984.17} C_VEL
LIN {X 0,Y 560.123,Z 554.681,A -85,B 0,C 180,E1 -2985.1,E2 -2985.1} C_VEL
LIN {X 0,Y 560.361,Z 541.502,A -85,B 0,C 180,E1 -2985.924,E2 -2985.924} C_VEL
LIN {X 0,Y 560.668,Z 526.816,A -85,B 0,C 180,E1 -2986.663,E2 -2986.663} C_VEL
LIN {X 0,Y 560.925,Z 512.602,A -85,B 0,C 180,E1 -2987.218,E2 -2987.218} C_VEL
LIN {X 0,Y 561.145,Z 498.127,A -85,B 0,C 180,E1 -2987.638,E2 -2987.638} C_VEL
LIN {X 0,Y 561.236,Z 483.608,A -85,B 0,C 180,E1 -2987.923,E2 -2987.923} C_VEL
LIN {X 0,Y 561.846,Z 330.01,A -85,B 0,C 180,E1 -2989.944,E2 -2989.944} C_VEL
LIN {X 0,Y 560.264,Z 321.655,A -85,B 0,C 180,E1 -2990.126,E2 -2990.126} C_VEL
LIN {X 0,Y 560.677,Z 297.007,A -85,B 0,C 180,E1 -2993.062,E2 -2993.062} C_VEL
LIN {X 0,Y 561.083,Z 272.715,A -85,B 0,C 180,E1 -2996.002,E2 -2996.002} C_VEL
LIN {X 0,Y 559.187,Z 263.456,A -85,B 0,C 180,E1 -2997.25,E2 -2997.25} C_VEL
LIN {X 0,Y 559.155,Z 263.46,A -85,B 0,C 180,E1 -3000.183,E2 -3000.183} C_VEL
LIN {X 0,Y 559.155,Z 263.462,A -85,B 0,C 180,E1 -3002.716,E2 -3002.716} C_VEL
LIN {X 0,Y 559.13,Z 263.458,A -85,B 0,C 180,E1 -3005.324,E2 -3005.324} C_VEL
LIN {X 0,Y 559.135,Z 263.459,A -85,B 0,C 180,E1 -3008.018,E2 -3008.018} C_VEL
LIN {X 0,Y 559.158,Z 263.458,A -85,B 0,C 180,E1 -3010.813,E2 -3010.813} C_VEL
LIN {X 0,Y 559.113,Z 263.46,A -85,B 0,C 180,E1 -3013.737,E2 -3013.737} C_VEL
LIN {X 0,Y 559.141,Z 263.463,A -85,B 0,C 180,E1 -3016.266,E2 -3016.266} C_VEL
LIN {X 0,Y 559.158,Z 263.454,A -85,B 0,C 180,E1 -3019.188,E2 -3019.188} C_VEL
LIN {X 0,Y 559.132,Z 263.461,A -85,B 0,C 180,E1 -3021.982,E2 -3021.982} C_VEL
LIN {X 0,Y 559.128,Z 263.459,A -85,B 0,C 180,E1 -3024.789,E2 -3024.789} C_VEL
LIN {X 0,Y 559.158,Z 263.452,A -85,B 0,C 180,E1 -3027.365,E2 -3027.365} C_VEL
LIN {X 0,Y 559.151,Z 263.463,A -85,B 0,C 180,E1 -3030.143,E2 -3030.143} C_VEL
LIN {X 0,Y 559.124,Z 263.457,A -85,B 0,C 180,E1 -3033.183,E2 -3033.183} C_VEL
LIN {X 0,Y 559.158,Z 263.454,A -85,B 0,C 180,E1 -3035.495,E2 -3035.495} C_VEL
LIN {X 0,Y 559.177,Z 263.453,A -85,B 0,C 180,E1 -3038.624,E2 -3038.624} C_VEL
LIN {X 0,Y 559.163,Z 263.452,A -85,B 0,C 180,E1 -3040.926,E2 -3040.926} C_VEL
LIN {X 0,Y 559.158,Z 263.462,A -85,B 0,C 180,E1 -3043.948,E2 -3043.948} C_VEL
LIN {X 0,Y 559.169,Z 263.459,A -85,B 0,C 180,E1 -3046.184,E2 -3046.184} C_VEL
LIN {X 0,Y 559.196,Z 263.448,A -85,B 0,C 180,E1 -3049.134,E2 -3049.134} C_VEL
LIN {X 0,Y 559.148,Z 263.461,A -85,B 0,C 180,E1 -3052.053,E2 -3052.053} C_VEL
LIN {X 0,Y 559.244,Z 263.443,A -85,B 0,C 180,E1 -3054.953,E2 -3054.953} C_VEL
LIN {X 0,Y 559.248,Z 263.45,A -85,B 0,C 180,E1 -3057.839,E2 -3057.839} C_VEL
LIN {X 0,Y 559.255,Z 263.448,A -85,B 0,C 180,E1 -3060,E2 -3060} C_VEL
LIN {X 0,Y 559.223,Z 263.445,A -85,B 0,C 180,E1 -3062.882,E2 -3062.882} C_VEL
LIN {X 0,Y 559.212,Z 263.455,A -85,B 0,C 180,E1 -3065.77,E2 -3065.77} C_VEL
LIN {X 0,Y 559.151,Z 263.454,A -85,B 0,C 180,E1 -3068.675,E2 -3068.675} C_VEL
LIN {X 0,Y 559.2,Z 263.455,A -85,B 0,C 180,E1 -3071.601,E2 -3071.601} C_VEL
LIN {X 0,Y 559.158,Z 263.452,A -85,B 0,C 180,E1 -3074.576,E2 -3074.576} C_VEL
LIN {X 0,Y 559.117,Z 263.468,A -85,B 0,C 180,E1 -3077.558,E2 -3077.558} C_VEL
LIN {X 0,Y 559.141,Z 263.462,A -85,B 0,C 180,E1 -3079.839,E2 -3079.839} C_VEL
LIN {X 0,Y 559.105,Z 263.461,A -85,B 0,C 180,E1 -3082.154,E2 -3082.154} C_VEL
LIN {X 0,Y 559.133,Z 263.461,A -85,B 0,C 180,E1 -3085.175,E2 -3085.175} C_VEL
LIN {X 0,Y 559.103,Z 263.462,A -85,B 0,C 180,E1 -3087.716,E2 -3087.716} C_VEL
LIN {X 0,Y 559.1,Z 263.46,A -85,B 0,C 180,E1 -3090.568,E2 -3090.568} C_VEL
LIN {X 0,Y 558.457,Z 263.548,A -85,B 0,C 180,E1 -3091.169,E2 -3091.169} C_VEL
LIN {X 0,Y 555.604,Z 263.899,A -85,B 0,C 180,E1 -3092.146,E2 -3092.146} C_VEL
LIN {X 0,Y 553.184,Z 264.2,A -85,B 0,C 180,E1 -3092.932,E2 -3092.932} C_VEL
LIN {X 0,Y 552.152,Z 264.334,A -85,B 0,C 180,E1 -3093.538,E2 -3093.538} C_VEL
LIN {X 0,Y 552.073,Z 264.337,A -85,B 0,C 180,E1 -3093.744,E2 -3093.744} C_VEL
LIN {X 0,Y 552.053,Z 264.339,A -85,B 0,C 180,E1 -3096.751,E2 -3096.751} C_VEL
LIN {X 0,Y 552.07,Z 264.343,A -85,B 0,C 180,E1 -3099.532,E2 -3099.532} C_VEL
LIN {X 0,Y 552.081,Z 264.335,A -85,B 0,C 180,E1 -3102.43,E2 -3102.43} C_VEL
LIN {X 0,Y 552.06,Z 264.342,A -85,B 0,C 180,E1 -3105.558,E2 -3105.558} C_VEL
LIN {X 0,Y 552.045,Z 264.341,A -85,B 0,C 180,E1 -3108.688,E2 -3108.688} C_VEL
LIN {X 0,Y 552.068,Z 264.343,A -85,B 0,C 180,E1 -3111.406,E2 -3111.406} C_VEL
LIN {X 0,Y 552.061,Z 264.34,A -85,B 0,C 180,E1 -3114.563,E2 -3114.563} C_VEL
LIN {X 0,Y 552.096,Z 264.343,A -85,B 0,C 180,E1 -3117.157,E2 -3117.157} C_VEL
LIN {X 0,Y 552.068,Z 264.338,A -85,B 0,C 180,E1 -3119.959,E2 -3119.959} C_VEL
LIN {X 0,Y 552.077,Z 264.344,A -85,B 0,C 180,E1 -3123.013,E2 -3123.013} C_VEL
LIN {X 0,Y 552.067,Z 264.342,A -85,B 0,C 180,E1 -3125.96,E2 -3125.96} C_VEL
LIN {X 0,Y 552.12,Z 264.434,A -85,B 0,C 180,E1 -3126.758,E2 -3126.758} C_VEL
LIN {X 0,Y 553.326,Z 271.361,A -85,B 0,C 180,E1 -3127.87,E2 -3127.87} C_VEL
LIN {X 0,Y 553.13,Z 283.397,A -85,B 0,C 180,E1 -3129.678,E2 -3129.678} C_VEL
LIN {X 0,Y 555.124,Z 293.596,A -85,B 0,C 180,E1 -3129.894,E2 -3129.894} C_VEL
LIN {X 0,Y 554.483,Z 448.306,A -85,B 0,C 180,E1 -3131.972,E2 -3131.972} C_VEL
LIN {X 0,Y 554.29,Z 463.793,A -85,B 0,C 180,E1 -3132.331,E2 -3132.331} C_VEL
LIN {X 0,Y 554.007,Z 479.093,A -85,B 0,C 180,E1 -3132.845,E2 -3132.845} C_VEL
LIN {X 0,Y 553.736,Z 493.742,A -85,B 0,C 180,E1 -3133.502,E2 -3133.502} C_VEL
LIN {X 0,Y 553.366,Z 507.062,A -85,B 0,C 180,E1 -3134.248,E2 -3134.248} C_VEL
LIN {X 0,Y 553.064,Z 520.724,A -85,B 0,C 180,E1 -3135.191,E2 -3135.191} C_VEL
LIN {X 0,Y 552.724,Z 532.899,A -85,B 0,C 180,E1 -3136.207,E2 -3136.207} C_VEL
LIN {X 0,Y 552.489,Z 544.092,A -85,B 0,C 180,E1 -3137.324,E2 -3137.324} C_VEL
LIN {X 0,Y 552.2,Z 555.339,A -85,B 0,C 180,E1 -3138.672,E2 -3138.672} C_VEL
LIN {X 0,Y 552.076,Z 564.008,A -85,B 0,C 180,E1 -3139.919,E2 -3139.919} C_VEL
LIN {X 0,Y 551.921,Z 571.497,A -85,B 0,C 180,E1 -3141.21,E2 -3141.21} C_VEL
LIN {X 0,Y 551.821,Z 578.502,A -85,B 0,C 180,E1 -3142.683,E2 -3142.683} C_VEL
LIN {X 0,Y 551.794,Z 584.012,A -85,B 0,C 180,E1 -3144.151,E2 -3144.151} C_VEL
LIN {X 0,Y 551.706,Z 588.178,A -85,B 0,C 180,E1 -3145.616,E2 -3145.616} C_VEL
LIN {X 0,Y 551.717,Z 591.112,A -85,B 0,C 180,E1 -3147.079,E2 -3147.079} C_VEL
LIN {X 0,Y 551.642,Z 592.878,A -85,B 0,C 180,E1 -3148.54,E2 -3148.54} C_VEL
LIN {X 0,Y 551.638,Z 593.496,A -85,B 0,C 180,E1 -3150,E2 -3150} C_VEL
LIN {X 0,Y 551.644,Z 592.94,A -85,B 0,C 180,E1 -3151.46,E2 -3151.46} C_VEL
LIN {X 0,Y 551.719,Z 591.255,A -85,B 0,C 180,E1 -3152.92,E2 -3152.92} C_VEL
LIN {X 0,Y 551.706,Z 588.402,A -85,B 0,C 180,E1 -3154.383,E2 -3154.383} C_VEL
LIN {X 0,Y 551.787,Z 584.315,A -85,B 0,C 180,E1 -3155.848,E2 -3155.848} C_VEL
LIN {X 0,Y 551.82,Z 578.899,A -85,B 0,C 180,E1 -3157.317,E2 -3157.317} C_VEL
LIN {X 0,Y 551.918,Z 571.997,A -85,B 0,C 180,E1 -3158.789,E2 -3158.789} C_VEL
LIN {X 0,Y 552.071,Z 564.571,A -85,B 0,C 180,E1 -3160.081,E2 -3160.081} C_VEL
LIN {X 0,Y 552.183,Z 556.06,A -85,B 0,C 180,E1 -3161.32,E2 -3161.32} C_VEL
LIN {X 0,Y 552.403,Z 546.533,A -85,B 0,C 180,E1 -3162.491,E2 -3162.491} C_VEL
LIN {X 0,Y 552.672,Z 535.799,A -85,B 0,C 180,E1 -3163.606,E2 -3163.606} C_VEL
LIN {X 0,Y 552.969,Z 524.087,A -85,B 0,C 180,E1 -3164.631,E2 -3164.631} C_VEL
LIN {X 0,Y 553.294,Z 511.302,A -85,B 0,C 180,E1 -3165.565,E2 -3165.565} C_VEL
LIN {X 0,Y 553.609,Z 498.971,A -85,B 0,C 180,E1 -3166.312,E2 -3166.312} C_VEL
LIN {X 0,Y 553.889,Z 484.629,A -85,B 0,C 180,E1 -3167.015,E2 -3167.015} C_VEL
LIN {X 0,Y 554.205,Z 469.731,A -85,B 0,C 180,E1 -3167.576,E2 -3167.576} C_VEL
LIN {X 0,Y 554.361,Z 454.662,A -85,B 0,C 180,E1 -3167.99,E2 -3167.99} C_VEL
LIN {X 0,Y 554.525,Z 439.384,A -85,B 0,C 180,E1 -3168.257,E2 -3168.257} C_VEL
LIN {X 0,Y 555.158,Z 293.227,A -85,B 0,C 180,E1 -3170.199,E2 -3170.199} C_VEL
LIN {X 0,Y 553.088,Z 283.336,A -85,B 0,C 180,E1 -3170.423,E2 -3170.423} C_VEL
LIN {X 0,Y 553.293,Z 270.185,A -85,B 0,C 180,E1 -3172.399,E2 -3172.399} C_VEL
LIN {X 0,Y 552.105,Z 264.341,A -85,B 0,C 180,E1 -3173.365,E2 -3173.365} C_VEL
LIN {X 0,Y 552.075,Z 264.34,A -85,B 0,C 180,E1 -3176.459,E2 -3176.459} C_VEL
LIN {X 0,Y 552.044,Z 264.349,A -85,B 0,C 180,E1 -3178.932,E2 -3178.932} C_VEL
LIN {X 0,Y 552.09,Z 264.339,A -85,B 0,C 180,E1 -3181.472,E2 -3181.472} C_VEL
LIN {X 0,Y 552.085,Z 264.337,A -85,B 0,C 180,E1 -3184.163,E2 -3184.163} C_VEL
LIN {X 0,Y 552.067,Z 264.343,A -85,B 0,C 180,E1 -3186.75,E2 -3186.75} C_VEL
LIN {X 0,Y 552.106,Z 264.334,A -85,B 0,C 180,E1 -3189.529,E2 -3189.529} C_VEL
LIN {X 0,Y 552.077,Z 264.339,A -85,B 0,C 180,E1 -3192.43,E2 -3192.43} C_VEL
LIN {X 0,Y 552.064,Z 264.338,A -85,B 0,C 180,E1 -3195.559,E2 -3195.559} C_VEL
LIN {X 0,Y 552.049,Z 264.341,A -85,B 0,C 180,E1 -3198.547,E2 -3198.547} C_VEL
LIN {X 0,Y 552.069,Z 264.337,A -85,B 0,C 180,E1 -3201.407,E2 -3201.407} C_VEL
LIN {X 0,Y 552.053,Z 264.341,A -85,B 0,C 180,E1 -3204.564,E2 -3204.564} C_VEL
LIN {X 0,Y 552.093,Z 264.336,A -85,B 0,C 180,E1 -3207.157,E2 -3207.157} C_VEL
LIN {X 0,Y 552.065,Z 264.338,A -85,B 0,C 180,E1 -3209.958,E2 -3209.958} C_VEL
LIN {X 0,Y 552.074,Z 264.339,A -85,B 0,C 180,E1 -3213.013,E2 -3213.013} C_VEL
LIN {X 0,Y 552.063,Z 264.339,A -85,B 0,C 180,E1 -3215.96,E2 -3215.96} C_VEL
LIN {X 0,Y 552.068,Z 264.338,A -85,B 0,C 180,E1 -3219.118,E2 -3219.118} C_VEL
LIN {X 0,Y 552.075,Z 264.334,A -85,B 0,C 180,E1 -3221.443,E2 -3221.443} C_VEL
LIN {X 0,Y 552.083,Z 264.342,A -85,B 0,C 180,E1 -3224.495,E2 -3224.495} C_VEL
LIN {X 0,Y 552.101,Z 264.332,A -85,B 0,C 180,E1 -3227.502,E2 -3227.502} C_VEL
LIN {X 0,Y 552.083,Z 264.336,A -85,B 0,C 180,E1 -3229.734,E2 -3229.734} C_VEL
LIN {X 0,Y 552.132,Z 264.331,A -85,B 0,C 180,E1 -3231.951,E2 -3231.951} C_VEL
LIN {X 0,Y 552.206,Z 264.319,A -85,B 0,C 180,E1 -3234.889,E2 -3234.889} C_VEL
LIN {X 0,Y 552.211,Z 264.322,A -85,B 0,C 180,E1 -3237.812,E2 -3237.812} C_VEL
LIN {X 0,Y 552.236,Z 264.315,A -85,B 0,C 180,E1 -3240.729,E2 -3240.729} C_VEL
LIN {X 0,Y 552.187,Z 264.323,A -85,B 0,C 180,E1 -3242.918,E2 -3242.918} C_VEL
LIN {X 0,Y 552.178,Z 264.327,A -85,B 0,C 180,E1 -3245.844,E2 -3245.844} C_VEL
LIN {X 0,Y 552.134,Z 264.329,A -85,B 0,C 180,E1 -3248.786,E2 -3248.786} C_VEL
LIN {X 0,Y 552.16,Z 264.328,A -85,B 0,C 180,E1 -3251.75,E2 -3251.75} C_VEL
LIN {X 0,Y 552.135,Z 264.327,A -85,B 0,C 180,E1 -3254.748,E2 -3254.748} C_VEL
LIN {X 0,Y 552.093,Z 264.341,A -85,B 0,C 180,E1 -3257.789,E2 -3257.789} C_VEL
LIN {X 0,Y 552.125,Z 264.337,A -85,B 0,C 180,E1 -3260.101,E2 -3260.101} C_VEL
LIN {X 0,Y 552.089,Z 264.336,A -85,B 0,C 180,E1 -3262.451,E2 -3262.451} C_VEL
LIN {X 0,Y 552.136,Z 264.325,A -85,B 0,C 180,E1 -3265.346,E2 -3265.346} C_VEL
LIN {X 0,Y 552.076,Z 264.341,A -85,B 0,C 180,E1 -3268.1,E2 -3268.1} C_VEL
LIN {X 0,Y 552.1,Z 264.331,A -85,B 0,C 180,E1 -3270.609,E2 -3270.609} C_VEL
LIN {X 0,Y 552.114,Z 264.33,A -85,B 0,C 180,E1 -3273.186,E2 -3273.186} C_VEL
LIN {X 0,Y 552.099,Z 264.339,A -85,B 0,C 180,E1 -3275.843,E2 -3275.843} C_VEL
LIN {X 0,Y 552.118,Z 264.331,A -85,B 0,C 180,E1 -3279.061,E2 -3279.061} C_VEL
LIN {X 0,Y 552.119,Z 264.337,A -85,B 0,C 180,E1 -3281.446,E2 -3281.446} C_VEL
LIN {X 0,Y 552.087,Z 264.335,A -85,B 0,C 180,E1 -3284.531,E2 -3284.531} C_VEL
LIN {X 0,Y 552.128,Z 264.338,A -85,B 0,C 180,E1 -3287.585,E2 -3287.585} C_VEL
LIN {X 0,Y 552.128,Z 264.33,A -85,B 0,C 180,E1 -3290.473,E2 -3290.473} C_VEL
LIN {X 0,Y 552.111,Z 264.338,A -85,B 0,C 180,E1 -3293.316,E2 -3293.316} C_VEL
LIN {X 0,Y 552.128,Z 264.333,A -85,B 0,C 180,E1 -3295.939,E2 -3295.939} C_VEL
LIN {X 0,Y 552.118,Z 264.332,A -85,B 0,C 180,E1 -3298.541,E2 -3298.541} C_VEL
LIN {X 0,Y 552.124,Z 264.339,A -85,B 0,C 180,E1 -3301.438,E2 -3301.438} C_VEL
LIN {X 0,Y 552.172,Z 264.475,A -85,B 0,C 180,E1 -3302.549,E2 -3302.549} C_VEL
LIN {X 0,Y 554.213,Z 273.986,A -85,B 0,C 180,E1 -3303.841,E2 -3303.841} C_VEL
LIN {X 0,Y 553.858,Z 295.138,A -85,B 0,C 180,E1 -3306.44,E2 -3306.44} C_VEL
LIN {X 0,Y 553.36,Z 321.536,A -85,B 0,C 180,E1 -3309.617,E2 -3309.617} C_VEL
LIN {X 0,Y 555.172,Z 332.122,A -85,B 0,C 180,E1 -3309.835,E2 -3309.835} C_VEL
LIN {X 0,Y 554.488,Z 487.739,A -85,B 0,C 180,E1 -3311.917,E2 -3311.917} C_VEL
LIN {X 0,Y 554.304,Z 503.711,A -85,B 0,C 180,E1 -3312.285,E2 -3312.285} C_VEL
LIN {X 0,Y 554.014,Z 519.041,A -85,B 0,C 180,E1 -3312.799,E2 -3312.799} C_VEL
LIN {X 0,Y 553.773,Z 532.786,A -85,B 0,C 180,E1 -3313.409,E2 -3313.409} C_VEL
LIN {X 0,Y 553.405,Z 546.258,A -85,B 0,C 180,E1 -3314.155,E2 -3314.155} C_VEL
LIN {X 0,Y 553.08,Z 560.132,A -85,B 0,C 180,E1 -3315.102,E2 -3315.102} C_VEL
LIN {X 0,Y 552.76,Z 572.357,A -85,B 0,C 180,E1 -3316.115,E2 -3316.115} C_VEL
LIN {X 0,Y 552.482,Z 584.511,A -85,B 0,C 180,E1 -3317.325,E2 -3317.325} C_VEL
LIN {X 0,Y 552.215,Z 594.486,A -85,B 0,C 180,E1 -3318.514,E2 -3318.514} C_VEL
LIN {X 0,Y 552.124,Z 603.088,A -85,B 0,C 180,E1 -3319.735,E2 -3319.735} C_VEL
LIN {X 0,Y 551.921,Z 610.744,A -85,B 0,C 180,E1 -3321.026,E2 -3321.026} C_VEL
LIN {X 0,Y 551.837,Z 617.091,A -85,B 0,C 180,E1 -3322.315,E2 -3322.315} C_VEL
LIN {X 0,Y 551.758,Z 622.608,A -85,B 0,C 180,E1 -3323.692,E2 -3323.692} C_VEL
LIN {X 0,Y 551.713,Z 626.388,A -85,B 0,C 180,E1 -3324.884,E2 -3324.884} C_VEL
LIN {X 0,Y 551.73,Z 629.889,A -85,B 0,C 180,E1 -3326.349,E2 -3326.349} C_VEL
LIN {X 0,Y 551.654,Z 632.191,A -85,B 0,C 180,E1 -3327.81,E2 -3327.81} C_VEL
LIN {X 0,Y 551.639,Z 633.348,A -85,B 0,C 180,E1 -3329.27,E2 -3329.27} C_VEL
LIN {X 0,Y 551.639,Z 633.348,A -85,B 0,C 180,E1 -3330.73,E2 -3330.73} C_VEL
LIN {X 0,Y 551.654,Z 632.187,A -85,B 0,C 180,E1 -3332.191,E2 -3332.191} C_VEL
LIN {X 0,Y 551.73,Z 629.884,A -85,B 0,C 180,E1 -3333.652,E2 -3333.652} C_VEL
LIN {X 0,Y 551.713,Z 626.386,A -85,B 0,C 180,E1 -3335.116,E2 -3335.116} C_VEL
LIN {X 0,Y 551.78,Z 621.607,A -85,B 0,C 180,E1 -3336.583,E2 -3336.583} C_VEL
LIN {X 0,Y 551.876,Z 615.419,A -85,B 0,C 180,E1 -3338.053,E2 -3338.053} C_VEL
LIN {X 0,Y 551.951,Z 607.642,A -85,B 0,C 180,E1 -3339.528,E2 -3339.528} C_VEL
LIN {X 0,Y 552.184,Z 599.365,A -85,B 0,C 180,E1 -3340.821,E2 -3340.821} C_VEL
LIN {X 0,Y 552.353,Z 589.388,A -85,B 0,C 180,E1 -3342.119,E2 -3342.119} C_VEL
LIN {X 0,Y 552.609,Z 579.181,A -85,B 0,C 180,E1 -3343.234,E2 -3343.234} C_VEL
LIN {X 0,Y 552.89,Z 567.014,A -85,B 0,C 180,E1 -3344.352,E2 -3344.352} C_VEL
LIN {X 0,Y 553.264,Z 554.435,A -85,B 0,C 180,E1 -3345.31,E2 -3345.31} C_VEL
LIN {X 0,Y 553.514,Z 541.499,A -85,B 0,C 180,E1 -3346.126,E2 -3346.126} C_VEL
LIN {X 0,Y 553.867,Z 526.813,A -85,B 0,C 180,E1 -3346.874,E2 -3346.874} C_VEL
LIN {X 0,Y 554.143,Z 512.602,A -85,B 0,C 180,E1 -3347.436,E2 -3347.436} C_VEL
LIN {X 0,Y 554.401,Z 497.489,A -85,B 0,C 180,E1 -3347.876,E2 -3347.876} C_VEL
LIN {X 0,Y 554.509,Z 483.273,A -85,B 0,C 180,E1 -3348.154,E2 -3348.154} C_VEL
LIN {X 0,Y 555.064,Z 330.351,A -85,B 0,C 180,E1 -3350.193,E2 -3350.193} C_VEL
LIN {X 0,Y 553.342,Z 321.515,A -85,B 0,C 180,E1 -3350.386,E2 -3350.386} C_VEL
LIN {X 0,Y 553.862,Z 295.132,A -85,B 0,C 180,E1 -3353.56,E2 -3353.56} C_VEL
LIN {X 0,Y 554.226,Z 273.84,A -85,B 0,C 180,E1 -3356.176,E2 -3356.176} C_VEL
LIN {X 0,Y 552.144,Z 264.333,A -85,B 0,C 180,E1 -3357.479,E2 -3357.479} C_VEL
LIN {X 0,Y 552.104,Z 264.34,A -85,B 0,C 180,E1 -3360.61,E2 -3360.61} C_VEL
LIN {X 0,Y 552.115,Z 264.334,A -85,B 0,C 180,E1 -3363.186,E2 -3363.186} C_VEL
LIN {X 0,Y 552.089,Z 264.336,A -85,B 0,C 180,E1 -3365.844,E2 -3365.844} C_VEL
LIN {X 0,Y 552.119,Z 264.336,A -85,B 0,C 180,E1 -3368.589,E2 -3368.589} C_VEL
LIN {X 0,Y 552.123,Z 264.33,A -85,B 0,C 180,E1 -3371.446,E2 -3371.446} C_VEL
LIN {X 0,Y 552.079,Z 264.343,A -85,B 0,C 180,E1 -3374.53,E2 -3374.53} C_VEL
LIN {X 0,Y 552.133,Z 264.328,A -85,B 0,C 180,E1 -3377.585,E2 -3377.585} C_VEL
LIN {X 0,Y 552.131,Z 264.336,A -85,B 0,C 180,E1 -3380.473,E2 -3380.473} C_VEL
LIN {X 0,Y 552.101,Z 264.332,A -85,B 0,C 180,E1 -3383.319,E2 -3383.319} C_VEL
LIN {X 0,Y 552.128,Z 264.333,A -85,B 0,C 180,E1 -3385.939,E2 -3385.939} C_VEL
LIN {X 0,Y 552.124,Z 264.334,A -85,B 0,C 180,E1 -3388.541,E2 -3388.541} C_VEL
LIN {X 0,Y 552.101,Z 264.332,A -85,B 0,C 180,E1 -3391.444,E2 -3391.444} C_VEL
LIN {X 0,Y 552.126,Z 264.331,A -85,B 0,C 180,E1 -3394.658,E2 -3394.658} C_VEL
LIN {X 0,Y 552.095,Z 264.334,A -85,B 0,C 180,E1 -3397.549,E2 -3397.549} C_VEL
LIN {X 0,Y 552.149,Z 264.33,A -85,B 0,C 180,E1 -3400.375,E2 -3400.375} C_VEL
LIN {X 0,Y 552.127,Z 264.329,A -85,B 0,C 180,E1 -3402.976,E2 -3402.976} C_VEL
LIN {X 0,Y 552.136,Z 264.337,A -85,B 0,C 180,E1 -3406.005,E2 -3406.005} C_VEL
LIN {X 0,Y 552.165,Z 264.323,A -85,B 0,C 180,E1 -3408.994,E2 -3408.994} C_VEL
LIN {X 0,Y 552.117,Z 264.339,A -85,B 0,C 180,E1 -3411.951,E2 -3411.951} C_VEL
LIN {X 0,Y 552.219,Z 264.318,A -85,B 0,C 180,E1 -3414.889,E2 -3414.889} C_VEL
LIN {X 0,Y 552.22,Z 264.325,A -85,B 0,C 180,E1 -3417.812,E2 -3417.812} C_VEL
LIN {X 0,Y 552.224,Z 264.324,A -85,B 0,C 180,E1 -3420,E2 -3420} C_VEL
LIN {X 0,Y 552.191,Z 264.321,A -85,B 0,C 180,E1 -3422.918,E2 -3422.918} C_VEL
LIN {X 0,Y 552.18,Z 264.33,A -85,B 0,C 180,E1 -3425.844,E2 -3425.844} C_VEL
LIN {X 0,Y 552.125,Z 264.33,A -85,B 0,C 180,E1 -3428.786,E2 -3428.786} C_VEL
LIN {X 0,Y 552.154,Z 264.335,A -85,B 0,C 180,E1 -3431.751,E2 -3431.751} C_VEL
LIN {X 0,Y 552.124,Z 264.328,A -85,B 0,C 180,E1 -3434.749,E2 -3434.749} C_VEL
LIN {X 0,Y 552.079,Z 264.341,A -85,B 0,C 180,E1 -3437.79,E2 -3437.79} C_VEL
LIN {X 0,Y 552.096,Z 264.336,A -85,B 0,C 180,E1 -3440.103,E2 -3440.103} C_VEL
LIN {X 0,Y 552.045,Z 264.338,A -85,B 0,C 180,E1 -3442.453,E2 -3442.453} C_VEL
LIN {X 0,Y 552.076,Z 264.342,A -85,B 0,C 180,E1 -3445.331,E2 -3445.331} C_VEL
LIN {X 0,Y 552.051,Z 264.336,A -85,B 0,C 180,E1 -3448.102,E2 -3448.102} C_VEL
LIN {X 0,Y 552.07,Z 264.336,A -85,B 0,C 180,E1 -3450.611,E2 -3450.611} C_VEL
LIN {X 0,Y 552.091,Z 264.339,A -85,B 0,C 180,E1 -3453.188,E2 -3453.188} C_VEL
LIN {X 0,Y 552.073,Z 264.337,A -85,B 0,C 180,E1 -3453.744,E2 -3453.744} C_VEL
LIN {X 0,Y 551.416,Z 264.421,A -85,B 0,C 180,E1 -3454.353,E2 -3454.353} C_VEL
LIN {X 0,Y 548.554,Z 264.784,A -85,B 0,C 180,E1 -3455.341,E2 -3455.341} C_VEL
LIN {X 0,Y 546.127,Z 265.08,A -85,B 0,C 180,E1 -3456.136,E2 -3456.136} C_VEL
LIN {X 0,Y 545.085,Z 265.208,A -85,B 0,C 180,E1 -3456.751,E2 -3456.751} C_VEL
LIN {X 0,Y 545,Z 265.22,A -85,B 0,C 180,E1 -3456.959,E2 -3456.959} C_VEL
LIN {X 0,Y 545.021,Z 265.222,A -85,B 0,C 180,E1 -3459.312,E2 -3459.312} C_VEL
LIN {X 0,Y 545.03,Z 265.214,A -85,B 0,C 180,E1 -3462.108,E2 -3462.108} C_VEL
LIN {X 0,Y 545.011,Z 265.223,A -85,B 0,C 180,E1 -3465.173,E2 -3465.173} C_VEL
LIN {X 0,Y 545.013,Z 265.215,A -85,B 0,C 180,E1 -3468.41,E2 -3468.41} C_VEL
LIN {X 0,Y 545.028,Z 265.217,A -85,B 0,C 180,E1 -3470.813,E2 -3470.813} C_VEL
LIN {X 0,Y 545.001,Z 265.221,A -85,B 0,C 180,E1 -3473.616,E2 -3473.616} C_VEL
LIN {X 0,Y 545.031,Z 265.213,A -85,B 0,C 180,E1 -3476.325,E2 -3476.325} C_VEL
LIN {X 0,Y 545.033,Z 265.219,A -85,B 0,C 180,E1 -3478.95,E2 -3478.95} C_VEL
LIN {X 0,Y 545.034,Z 265.218,A -85,B 0,C 180,E1 -3481.503,E2 -3481.503} C_VEL
LIN {X 0,Y 545.018,Z 265.218,A -85,B 0,C 180,E1 -3483.996,E2 -3483.996} C_VEL
LIN {X 0,Y 545.088,Z 265.32,A -85,B 0,C 180,E1 -3486.541,E2 -3486.541} C_VEL
LIN {X 0,Y 546.472,Z 273.137,A -85,B 0,C 180,E1 -3487.815,E2 -3487.815} C_VEL
LIN {X 0,Y 546.281,Z 283.837,A -85,B 0,C 180,E1 -3489.414,E2 -3489.414} C_VEL
LIN {X 0,Y 548.466,Z 293.911,A -85,B 0,C 180,E1 -3489.64,E2 -3489.64} C_VEL
LIN {X 0,Y 547.745,Z 448.619,A -85,B 0,C 180,E1 -3491.743,E2 -3491.743} C_VEL
LIN {X 0,Y 547.529,Z 464.029,A -85,B 0,C 180,E1 -3492.105,E2 -3492.105} C_VEL
LIN {X 0,Y 547.262,Z 478.06,A -85,B 0,C 180,E1 -3492.579,E2 -3492.579} C_VEL
LIN {X 0,Y 546.955,Z 491.959,A -85,B 0,C 180,E1 -3493.195,E2 -3493.195} C_VEL
LIN {X 0,Y 546.552,Z 505.559,A -85,B 0,C 180,E1 -3493.95,E2 -3493.95} C_VEL
LIN {X 0,Y 546.212,Z 519.099,A -85,B 0,C 180,E1 -3494.878,E2 -3494.878} C_VEL
LIN {X 0,Y 545.876,Z 530.783,A -85,B 0,C 180,E1 -3495.84,E2 -3495.84} C_VEL
LIN {X 0,Y 545.573,Z 542.319,A -85,B 0,C 180,E1 -3496.971,E2 -3496.971} C_VEL
LIN {X 0,Y 545.289,Z 552.031,A -85,B 0,C 180,E1 -3498.099,E2 -3498.099} C_VEL
LIN {X 0,Y 545.09,Z 561.554,A -85,B 0,C 180,E1 -3499.413,E2 -3499.413} C_VEL
LIN {X 0,Y 544.878,Z 570.492,A -85,B 0,C 180,E1 -3500.909,E2 -3500.909} C_VEL
LIN {X 0,Y 544.774,Z 576.891,A -85,B 0,C 180,E1 -3502.215,E2 -3502.215} C_VEL
LIN {X 0,Y 544.676,Z 582.016,A -85,B 0,C 180,E1 -3503.483,E2 -3503.483} C_VEL
LIN {X 0,Y 544.642,Z 586.257,A -85,B 0,C 180,E1 -3504.817,E2 -3504.817} C_VEL
LIN {X 0,Y 544.645,Z 589.795,A -85,B 0,C 180,E1 -3506.3,E2 -3506.3} C_VEL
LIN {X 0,Y 544.569,Z 592.137,A -85,B 0,C 180,E1 -3507.781,E2 -3507.781} C_VEL
LIN {X 0,Y 544.537,Z 593.337,A -85,B 0,C 180,E1 -3509.26,E2 -3509.26} C_VEL
LIN {X 0,Y 544.538,Z 593.358,A -85,B 0,C 180,E1 -3510.739,E2 -3510.739} C_VEL
LIN {X 0,Y 544.57,Z 592.239,A -85,B 0,C 180,E1 -3512.219,E2 -3512.219} C_VEL
LIN {X 0,Y 544.646,Z 589.976,A -85,B 0,C 180,E1 -3513.699,E2 -3513.699} C_VEL
LIN {X 0,Y 544.641,Z 586.516,A -85,B 0,C 180,E1 -3515.182,E2 -3515.182} C_VEL
LIN {X 0,Y 544.698,Z 581.779,A -85,B 0,C 180,E1 -3516.668,E2 -3516.668} C_VEL
LIN {X 0,Y 544.819,Z 575.643,A -85,B 0,C 180,E1 -3518.157,E2 -3518.157} C_VEL
LIN {X 0,Y 544.903,Z 567.918,A -85,B 0,C 180,E1 -3519.652,E2 -3519.652} C_VEL
LIN {X 0,Y 545.128,Z 559.681,A -85,B 0,C 180,E1 -3520.962,E2 -3520.962} C_VEL
LIN {X 0,Y 545.332,Z 549.769,A -85,B 0,C 180,E1 -3522.277,E2 -3522.277} C_VEL
LIN {X 0,Y 545.617,Z 539.608,A -85,B 0,C 180,E1 -3523.406,E2 -3523.406} C_VEL
LIN {X 0,Y 545.922,Z 527.519,A -85,B 0,C 180,E1 -3524.538,E2 -3524.538} C_VEL
LIN {X 0,Y 546.374,Z 514.039,A -85,B 0,C 180,E1 -3525.582,E2 -3525.582} C_VEL
LIN {X 0,Y 546.749,Z 500.757,A -85,B 0,C 180,E1 -3526.427,E2 -3526.427} C_VEL
LIN {X 0,Y 547.083,Z 485.884,A -85,B 0,C 180,E1 -3527.185,E2 -3527.185} C_VEL
LIN {X 0,Y 547.415,Z 471.399,A -85,B 0,C 180,E1 -3527.753,E2 -3527.753} C_VEL
LIN {X 0,Y 547.64,Z 455.793,A -85,B 0,C 180,E1 -3528.198,E2 -3528.198} C_VEL
LIN {X 0,Y 547.801,Z 440.382,A -85,B 0,C 180,E1 -3528.479,E2 -3528.479} C_VEL
LIN {X 0,Y 548.485,Z 294.557,A -85,B 0,C 180,E1 -3530.441,E2 -3530.441} C_VEL
LIN {X 0,Y 546.239,Z 283.607,A -85,B 0,C 180,E1 -3530.69,E2 -3530.69} C_VEL
LIN {X 0,Y 546.376,Z 271.471,A -85,B 0,C 180,E1 -3532.536,E2 -3532.536} C_VEL
LIN {X 0,Y 545.054,Z 265.218,A -85,B 0,C 180,E1 -3533.6,E2 -3533.6} C_VEL
LIN {X 0,Y 545.037,Z 265.215,A -85,B 0,C 180,E1 -3536.002,E2 -3536.002} C_VEL
LIN {X 0,Y 545.022,Z 265.222,A -85,B 0,C 180,E1 -3538.735,E2 -3538.735} C_VEL
LIN {X 0,Y 545.042,Z 265.216,A -85,B 0,C 180,E1 -3541.676,E2 -3541.676} C_VEL
LIN {X 0,Y 545.04,Z 265.218,A -85,B 0,C 180,E1 -3544.566,E2 -3544.566} C_VEL
LIN {X 0,Y 545.014,Z 265.22,A -85,B 0,C 180,E1 -3547.305,E2 -3547.305} C_VEL
LIN {X 0,Y 545.052,Z 265.212,A -85,B 0,C 180,E1 -3550.144,E2 -3550.144} C_VEL
LIN {X 0,Y 544.996,Z 265.221,A -85,B 0,C 180,E1 -3553.114,E2 -3553.114} C_VEL
LIN {X 0,Y 545.023,Z 265.215,A -85,B 0,C 180,E1 -3555.867,E2 -3555.867} C_VEL
LIN {X 0,Y 544.993,Z 265.225,A -85,B 0,C 180,E1 -3558.877,E2 -3558.877} C_VEL
LIN {X 0,Y 545.016,Z 265.215,A -85,B 0,C 180,E1 -3561.868,E2 -3561.868} C_VEL
LIN {X 0,Y 545.013,Z 265.216,A -85,B 0,C 180,E1 -3564.53,E2 -3564.53} C_VEL
LIN {X 0,Y 545.048,Z 265.213,A -85,B 0,C 180,E1 -3567.21,E2 -3567.21} C_VEL
LIN {X 0,Y 545.015,Z 265.215,A -85,B 0,C 180,E1 -3569.807,E2 -3569.807} C_VEL
LIN {X 0,Y 544.995,Z 265.224,A -85,B 0,C 180,E1 -3572.339,E2 -3572.339} C_VEL
LIN {X 0,Y 545.033,Z 265.218,A -85,B 0,C 180,E1 -3574.816,E2 -3574.816} C_VEL
LIN {X 0,Y 544.985,Z 265.219,A -85,B 0,C 180,E1 -3577.24,E2 -3577.24} C_VEL
LIN {X 0,Y 545.099,Z 265.213,A -85,B 0,C 180,E1 -3580.414,E2 -3580.414} C_VEL
LIN {X 0,Y 545.014,Z 265.216,A -85,B 0,C 180,E1 -3583.519,E2 -3583.519} C_VEL
LIN {X 0,Y 545.058,Z 265.21,A -85,B 0,C 180,E1 -3585.819,E2 -3585.819} C_VEL
LIN {X 0,Y 545.109,Z 265.206,A -85,B 0,C 180,E1 -3588.849,E2 -3588.849} C_VEL
LIN {X 0,Y 545.083,Z 265.208,A -85,B 0,C 180,E1 -3591.846,E2 -3591.846} C_VEL
LIN {X 0,Y 545.164,Z 265.197,A -85,B 0,C 180,E1 -3594.822,E2 -3594.822} C_VEL
LIN {X 0,Y 545.184,Z 265.197,A -85,B 0,C 180,E1 -3597.784,E2 -3597.784} C_VEL
LIN {X 0,Y 545.206,Z 265.191,A -85,B 0,C 180,E1 -3600.739,E2 -3600.739} C_VEL
LIN {X 0,Y 545.153,Z 265.199,A -85,B 0,C 180,E1 -3602.956,E2 -3602.956} C_VEL
LIN {X 0,Y 545.128,Z 265.206,A -85,B 0,C 180,E1 -3605.92,E2 -3605.92} C_VEL
LIN {X 0,Y 545.095,Z 265.206,A -85,B 0,C 180,E1 -3608.9,E2 -3608.9} C_VEL
LIN {X 0,Y 545.103,Z 265.21,A -85,B 0,C 180,E1 -3611.905,E2 -3611.905} C_VEL
LIN {X 0,Y 545.084,Z 265.205,A -85,B 0,C 180,E1 -3614.944,E2 -3614.944} C_VEL
LIN {X 0,Y 545.059,Z 265.218,A -85,B 0,C 180,E1 -3618.026,E2 -3618.026} C_VEL
LIN {X 0,Y 545.09,Z 265.21,A -85,B 0,C 180,E1 -3620.372,E2 -3620.372} C_VEL
LIN {X 0,Y 545.077,Z 265.211,A -85,B 0,C 180,E1 -3623.559,E2 -3623.559} C_VEL
LIN {X 0,Y 545.072,Z 265.212,A -85,B 0,C 180,E1 -3626.001,E2 -3626.001} C_VEL
LIN {X 0,Y 545.067,Z 265.209,A -85,B 0,C 180,E1 -3628.744,E2 -3628.744} C_VEL
LIN {X 0,Y 545.057,Z 265.214,A -85,B 0,C 180,E1 -3631.679,E2 -3631.679} C_VEL
LIN {X 0,Y 545.065,Z 265.21,A -85,B 0,C 180,E1 -3634.564,E2 -3634.564} C_VEL
LIN {X 0,Y 545.036,Z 265.214,A -85,B 0,C 180,E1 -3637.304,E2 -3637.304} C_VEL
LIN {X 0,Y 545.063,Z 265.212,A -85,B 0,C 180,E1 -3640.143,E2 -3640.143} C_VEL
LIN {X 0,Y 545.077,Z 265.21,A -85,B 0,C 180,E1 -3643.107,E2 -3643.107} C_VEL
LIN {X 0,Y 545.047,Z 265.212,A -85,B 0,C 180,E1 -3646.226,E2 -3646.226} C_VEL
LIN {X 0,Y 545.081,Z 265.207,A -85,B 0,C 180,E1 -3648.886,E2 -3648.886} C_VEL
LIN {X 0,Y 545.051,Z 265.217,A -85,B 0,C 180,E1 -3651.763,E2 -3651.763} C_VEL
LIN {X 0,Y 545.052,Z 265.212,A -85,B 0,C 180,E1 -3654.533,E2 -3654.533} C_VEL
LIN {X 0,Y 545.068,Z 265.215,A -85,B 0,C 180,E1 -3657.212,E2 -3657.212} C_VEL
LIN {X 0,Y 545.063,Z 265.216,A -85,B 0,C 180,E1 -3659.811,E2 -3659.811} C_VEL
LIN {X 0,Y 545.103,Z 265.236,A -85,B 0,C 180,E1 -3662.293,E2 -3662.293} C_VEL
LIN {X 0,Y 547.355,Z 275.461,A -85,B 0,C 180,E1 -3663.707,E2 -3663.707} C_VEL
LIN {X 0,Y 546.993,Z 296.666,A -85,B 0,C 180,E1 -3666.348,E2 -3666.348} C_VEL
LIN {X 0,Y 546.439,Z 321.308,A -85,B 0,C 180,E1 -3669.351,E2 -3669.351} C_VEL
LIN {X 0,Y 548.482,Z 332.246,A -85,B 0,C 180,E1 -3669.584,E2 -3669.584} C_VEL
LIN {X 0,Y 547.742,Z 487.466,A -85,B 0,C 180,E1 -3671.684,E2 -3671.684} C_VEL
LIN {X 0,Y 547.542,Z 502.865,A -85,B 0,C 180,E1 -3672.037,E2 -3672.037} C_VEL
LIN {X 0,Y 547.253,Z 517.754,A -85,B 0,C 180,E1 -3672.531,E2 -3672.531} C_VEL
LIN {X 0,Y 546.954,Z 530.8,A -85,B 0,C 180,E1 -3673.099,E2 -3673.099} C_VEL
LIN {X 0,Y 546.564,Z 544.677,A -85,B 0,C 180,E1 -3673.856,E2 -3673.856} C_VEL
LIN {X 0,Y 546.287,Z 556.605,A -85,B 0,C 180,E1 -3674.651,E2 -3674.651} C_VEL
LIN {X 0,Y 545.914,Z 569.154,A -85,B 0,C 180,E1 -3675.652,E2 -3675.652} C_VEL
LIN {X 0,Y 545.589,Z 580.968,A -85,B 0,C 180,E1 -3676.783,E2 -3676.783} C_VEL
LIN {X 0,Y 545.315,Z 590.906,A -85,B 0,C 180,E1 -3677.911,E2 -3677.911} C_VEL
LIN {X 0,Y 545.136,Z 600.625,A -85,B 0,C 180,E1 -3679.226,E2 -3679.226} C_VEL
LIN {X 0,Y 544.891,Z 608.727,A -85,B 0,C 180,E1 -3680.535,E2 -3680.535} C_VEL
LIN {X 0,Y 544.818,Z 615.425,A -85,B 0,C 180,E1 -3681.843,E2 -3681.843} C_VEL
LIN {X 0,Y 544.7,Z 622.094,A -85,B 0,C 180,E1 -3683.46,E2 -3683.46} C_VEL
LIN {X 0,Y 544.642,Z 626.387,A -85,B 0,C 180,E1 -3684.818,E2 -3684.818} C_VEL
LIN {X 0,Y 544.644,Z 629.888,A -85,B 0,C 180,E1 -3686.301,E2 -3686.301} C_VEL
LIN {X 0,Y 544.568,Z 632.19,A -85,B 0,C 180,E1 -3687.781,E2 -3687.781} C_VEL
LIN {X 0,Y 544.539,Z 633.348,A -85,B 0,C 180,E1 -3689.261,E2 -3689.261} C_VEL
LIN {X 0,Y 544.539,Z 633.347,A -85,B 0,C 180,E1 -3690.74,E2 -3690.74} C_VEL
LIN {X 0,Y 544.568,Z 632.186,A -85,B 0,C 180,E1 -3692.219,E2 -3692.219} C_VEL
LIN {X 0,Y 544.644,Z 629.883,A -85,B 0,C 180,E1 -3693.7,E2 -3693.7} C_VEL
LIN {X 0,Y 544.642,Z 626.386,A -85,B 0,C 180,E1 -3695.183,E2 -3695.183} C_VEL
LIN {X 0,Y 544.698,Z 621.608,A -85,B 0,C 180,E1 -3696.669,E2 -3696.669} C_VEL
LIN {X 0,Y 544.819,Z 615.418,A -85,B 0,C 180,E1 -3698.158,E2 -3698.158} C_VEL
LIN {X 0,Y 544.905,Z 607.641,A -85,B 0,C 180,E1 -3699.653,E2 -3699.653} C_VEL
LIN {X 0,Y 545.15,Z 599.364,A -85,B 0,C 180,E1 -3700.962,E2 -3700.962} C_VEL
LIN {X 0,Y 545.358,Z 589.388,A -85,B 0,C 180,E1 -3702.277,E2 -3702.277} C_VEL
LIN {X 0,Y 545.64,Z 579.18,A -85,B 0,C 180,E1 -3703.406,E2 -3703.406} C_VEL
LIN {X 0,Y 545.974,Z 567.013,A -85,B 0,C 180,E1 -3704.538,E2 -3704.538} C_VEL
LIN {X 0,Y 546.379,Z 553.375,A -85,B 0,C 180,E1 -3705.582,E2 -3705.582} C_VEL
LIN {X 0,Y 546.741,Z 539.873,A -85,B 0,C 180,E1 -3706.428,E2 -3706.428} C_VEL
LIN {X 0,Y 547.075,Z 525.768,A -85,B 0,C 180,E1 -3707.138,E2 -3707.138} C_VEL
LIN {X 0,Y 547.35,Z 511.217,A -85,B 0,C 180,E1 -3707.707,E2 -3707.707} C_VEL
LIN {X 0,Y 547.634,Z 495.802,A -85,B 0,C 180,E1 -3708.145,E2 -3708.145} C_VEL
LIN {X 0,Y 547.803,Z 480.5,A -85,B 0,C 180,E1 -3708.426,E2 -3708.426} C_VEL
LIN {X 0,Y 548.414,Z 331.462,A -85,B 0,C 180,E1 -3710.429,E2 -3710.429} C_VEL
LIN {X 0,Y 546.433,Z 321.252,A -85,B 0,C 180,E1 -3710.656,E2 -3710.656} C_VEL
LIN {X 0,Y 547,Z 296.66,A -85,B 0,C 180,E1 -3713.652,E2 -3713.652} C_VEL
LIN {X 0,Y 547.401,Z 275.452,A -85,B 0,C 180,E1 -3716.292,E2 -3716.292} C_VEL
LIN {X 0,Y 545.072,Z 265.215,A -85,B 0,C 180,E1 -3717.735,E2 -3717.735} C_VEL
LIN {X 0,Y 545.08,Z 265.214,A -85,B 0,C 180,E1 -3720.247,E2 -3720.247} C_VEL
LIN {X 0,Y 545.079,Z 265.211,A -85,B 0,C 180,E1 -3723.062,E2 -3723.062} C_VEL
LIN {X 0,Y 545.037,Z 265.214,A -85,B 0,C 180,E1 -3725.673,E2 -3725.673} C_VEL
LIN {X 0,Y 545.054,Z 265.216,A -85,B 0,C 180,E1 -3728.238,E2 -3728.238} C_VEL
LIN {X 0,Y 545.083,Z 265.215,A -85,B 0,C 180,E1 -3730.473,E2 -3730.473} C_VEL
LIN {X 0,Y 545.025,Z 265.215,A -85,B 0,C 180,E1 -3733.113,E2 -3733.113} C_VEL
LIN {X 0,Y 545.052,Z 265.217,A -85,B 0,C 180,E1 -3736.227,E2 -3736.227} C_VEL
LIN {X 0,Y 545.084,Z 265.209,A -85,B 0,C 180,E1 -3738.886,E2 -3738.886} C_VEL
LIN {X 0,Y 545.05,Z 265.214,A -85,B 0,C 180,E1 -3741.865,E2 -3741.865} C_VEL
LIN {X 0,Y 545.03,Z 265.218,A -85,B 0,C 180,E1 -3744.531,E2 -3744.531} C_VEL
LIN {X 0,Y 545.071,Z 265.207,A -85,B 0,C 180,E1 -3747.212,E2 -3747.212} C_VEL
LIN {X 0,Y 545.066,Z 265.212,A -85,B 0,C 180,E1 -3749.811,E2 -3749.811} C_VEL
LIN {X 0,Y 545.05,Z 265.217,A -85,B 0,C 180,E1 -3752.342,E2 -3752.342} C_VEL
LIN {X 0,Y 545.097,Z 265.206,A -85,B 0,C 180,E1 -3754.819,E2 -3754.819} C_VEL
LIN {X 0,Y 545.039,Z 265.211,A -85,B 0,C 180,E1 -3757.242,E2 -3757.242} C_VEL
LIN {X 0,Y 545.121,Z 265.205,A -85,B 0,C 180,E1 -3760.415,E2 -3760.415} C_VEL
LIN {X 0,Y 545.059,Z 265.212,A -85,B 0,C 180,E1 -3763.521,E2 -3763.521} C_VEL
LIN {X 0,Y 545.097,Z 265.21,A -85,B 0,C 180,E1 -3765.82,E2 -3765.82} C_VEL
LIN {X 0,Y 545.121,Z 265.201,A -85,B 0,C 180,E1 -3768.85,E2 -3768.85} C_VEL
LIN {X 0,Y 545.075,Z 265.216,A -85,B 0,C 180,E1 -3771.846,E2 -3771.846} C_VEL
LIN {X 0,Y 545.176,Z 265.195,A -85,B 0,C 180,E1 -3774.823,E2 -3774.823} C_VEL
LIN {X 0,Y 545.192,Z 265.2,A -85,B 0,C 180,E1 -3777.784,E2 -3777.784} C_VEL
LIN {X 0,Y 545.193,Z 265.2,A -85,B 0,C 180,E1 -3780,E2 -3780} C_VEL
LIN {X 0,Y 545.16,Z 265.197,A -85,B 0,C 180,E1 -3782.956,E2 -3782.956} C_VEL
LIN {X 0,Y 545.127,Z 265.207,A -85,B 0,C 180,E1 -3785.92,E2 -3785.92} C_VEL
LIN {X 0,Y 545.069,Z 265.209,A -85,B 0,C 180,E1 -3788.901,E2 -3788.901} C_VEL
LIN {X 0,Y 545.096,Z 265.212,A -85,B 0,C 180,E1 -3791.905,E2 -3791.905} C_VEL
LIN {X 0,Y 545.08,Z 265.206,A -85,B 0,C 180,E1 -3794.944,E2 -3794.944} C_VEL
LIN {X 0,Y 545.047,Z 265.213,A -85,B 0,C 180,E1 -3798.027,E2 -3798.027} C_VEL
LIN {X 0,Y 545.033,Z 265.214,A -85,B 0,C 180,E1 -3800.375,E2 -3800.375} C_VEL
LIN {X 0,Y 544.991,Z 265.217,A -85,B 0,C 180,E1 -3802.76,E2 -3802.76} C_VEL
LIN {X 0,Y 545.028,Z 265.223,A -85,B 0,C 180,E1 -3805.492,E2 -3805.492} C_VEL
LIN {X 0,Y 545.001,Z 265.218,A -85,B 0,C 180,E1 -3807.661,E2 -3807.661} C_VEL
LIN {X 0,Y 545.023,Z 265.215,A -85,B 0,C 180,E1 -3810.235,E2 -3810.235} C_VEL
LIN {X 0,Y 545.061,Z 265.213,A -85,B 0,C 180,E1 -3813.058,E2 -3813.058} C_VEL
LIN {X 0,Y 545.017,Z 265.22,A -85,B 0,C 180,E1 -3815.669,E2 -3815.669} C_VEL
LIN {X 0,Y 545,Z 265.22,A -85,B 0,C 180,E1 -3816.959,E2 -3816.959} C_VEL
LIN {X 0,Y 544.334,Z 265.309,A -85,B 0,C 180,E1 -3817.575,E2 -3817.575} C_VEL
LIN {X 0,Y 541.48,Z 265.664,A -85,B 0,C 180,E1 -3818.577,E2 -3818.577} C_VEL
LIN {X 0,Y 539.066,Z 265.965,A -85,B 0,C 180,E1 -3819.383,E2 -3819.383} C_VEL
LIN {X 0,Y 538.028,Z 266.087,A -85,B 0,C 180,E1 -3820.005,E2 -3820.005} C_VEL
LIN {X 0,Y 537.943,Z 266.096,A -85,B 0,C 180,E1 -3820.216,E2 -3820.216} C_VEL
LIN {X 0,Y 537.956,Z 266.099,A -85,B 0,C 180,E1 -3822.979,E2 -3822.979} C_VEL
LIN {X 0,Y 537.985,Z 266.098,A -85,B 0,C 180,E1 -3825.135,E2 -3825.135} C_VEL
LIN {X 0,Y 537.968,Z 266.093,A -85,B 0,C 180,E1 -3828.22,E2 -3828.22} C_VEL
LIN {X 0,Y 537.973,Z 266.102,A -85,B 0,C 180,E1 -3831.165,E2 -3831.165} C_VEL
LIN {X 0,Y 537.958,Z 266.096,A -85,B 0,C 180,E1 -3834.094,E2 -3834.094} C_VEL
LIN {X 0,Y 538.001,Z 266.092,A -85,B 0,C 180,E1 -3836.725,E2 -3836.725} C_VEL
LIN {X 0,Y 537.99,Z 266.095,A -85,B 0,C 180,E1 -3839.563,E2 -3839.563} C_VEL
LIN {X 0,Y 537.991,Z 266.096,A -85,B 0,C 180,E1 -3842.662,E2 -3842.662} C_VEL
LIN {X 0,Y 537.968,Z 266.102,A -85,B 0,C 180,E1 -3845.288,E2 -3845.288} C_VEL
LIN {X 0,Y 538.051,Z 266.249,A -85,B 0,C 180,E1 -3846.323,E2 -3846.323} C_VEL
LIN {X 0,Y 539.564,Z 274.171,A -85,B 0,C 180,E1 -3847.638,E2 -3847.638} C_VEL
LIN {X 0,Y 539.415,Z 283.93,A -85,B 0,C 180,E1 -3849.134,E2 -3849.134} C_VEL
LIN {X 0,Y 541.802,Z 294.656,A -85,B 0,C 180,E1 -3849.384,E2 -3849.384} C_VEL
LIN {X 0,Y 541.076,Z 443.673,A -85,B 0,C 180,E1 -3851.422,E2 -3851.422} C_VEL
LIN {X 0,Y 540.895,Z 457.892,A -85,B 0,C 180,E1 -3851.704,E2 -3851.704} C_VEL
LIN {X 0,Y 540.591,Z 473.168,A -85,B 0,C 180,E1 -3852.162,E2 -3852.162} C_VEL
LIN {X 0,Y 540.283,Z 486.292,A -85,B 0,C 180,E1 -3852.689,E2 -3852.689} C_VEL
LIN {X 0,Y 539.925,Z 501.115,A -85,B 0,C 180,E1 -3853.456,E2 -3853.456} C_VEL
LIN {X 0,Y 539.482,Z 514.477,A -85,B 0,C 180,E1 -3854.316,E2 -3854.316} C_VEL
LIN {X 0,Y 539.046,Z 527.787,A -85,B 0,C 180,E1 -3855.368,E2 -3855.368} C_VEL
LIN {X 0,Y 538.691,Z 538.88,A -85,B 0,C 180,E1 -3856.418,E2 -3856.418} C_VEL
LIN {X 0,Y 538.367,Z 549.05,A -85,B 0,C 180,E1 -3857.561,E2 -3857.561} C_VEL
LIN {X 0,Y 538.122,Z 559.044,A -85,B 0,C 180,E1 -3858.893,E2 -3858.893} C_VEL
LIN {X 0,Y 537.874,Z 567.375,A -85,B 0,C 180,E1 -3860.22,E2 -3860.22} C_VEL
LIN {X 0,Y 537.737,Z 575.202,A -85,B 0,C 180,E1 -3861.734,E2 -3861.734} C_VEL
LIN {X 0,Y 537.621,Z 581.438,A -85,B 0,C 180,E1 -3863.243,E2 -3863.243} C_VEL
LIN {X 0,Y 537.574,Z 586.258,A -85,B 0,C 180,E1 -3864.749,E2 -3864.749} C_VEL
LIN {X 0,Y 537.562,Z 589.795,A -85,B 0,C 180,E1 -3866.252,E2 -3866.252} C_VEL
LIN {X 0,Y 537.488,Z 592.137,A -85,B 0,C 180,E1 -3867.752,E2 -3867.752} C_VEL
LIN {X 0,Y 537.437,Z 593.337,A -85,B 0,C 180,E1 -3869.25,E2 -3869.25} C_VEL
LIN {X 0,Y 537.439,Z 593.357,A -85,B 0,C 180,E1 -3870.749,E2 -3870.749} C_VEL
LIN {X 0,Y 537.488,Z 592.237,A -85,B 0,C 180,E1 -3872.248,E2 -3872.248} C_VEL
LIN {X 0,Y 537.563,Z 589.974,A -85,B 0,C 180,E1 -3873.748,E2 -3873.748} C_VEL
LIN {X 0,Y 537.573,Z 586.514,A -85,B 0,C 180,E1 -3875.25,E2 -3875.25} C_VEL
LIN {X 0,Y 537.619,Z 581.776,A -85,B 0,C 180,E1 -3876.756,E2 -3876.756} C_VEL
LIN {X 0,Y 537.734,Z 575.639,A -85,B 0,C 180,E1 -3878.265,E2 -3878.265} C_VEL
LIN {X 0,Y 537.858,Z 567.914,A -85,B 0,C 180,E1 -3879.78,E2 -3879.78} C_VEL
LIN {X 0,Y 538.081,Z 559.677,A -85,B 0,C 180,E1 -3881.107,E2 -3881.107} C_VEL
LIN {X 0,Y 538.347,Z 549.803,A -85,B 0,C 180,E1 -3882.439,E2 -3882.439} C_VEL
LIN {X 0,Y 538.656,Z 539.721,A -85,B 0,C 180,E1 -3883.583,E2 -3883.583} C_VEL
LIN {X 0,Y 539.035,Z 527.715,A -85,B 0,C 180,E1 -3884.728,E2 -3884.728} C_VEL
LIN {X 0,Y 539.524,Z 514.416,A -85,B 0,C 180,E1 -3885.776,E2 -3885.776} C_VEL
LIN {X 0,Y 539.93,Z 501.018,A -85,B 0,C 180,E1 -3886.64,E2 -3886.64} C_VEL
LIN {X 0,Y 540.299,Z 486.141,A -85,B 0,C 180,E1 -3887.408,E2 -3887.408} C_VEL
LIN {X 0,Y 540.671,Z 471.651,A -85,B 0,C 180,E1 -3887.982,E2 -3887.982} C_VEL
LIN {X 0,Y 540.898,Z 455.999,A -85,B 0,C 180,E1 -3888.434,E2 -3888.434} C_VEL
LIN {X 0,Y 541.108,Z 439.556,A -85,B 0,C 180,E1 -3888.73,E2 -3888.73} C_VEL
LIN {X 0,Y 541.852,Z 295.423,A -85,B 0,C 180,E1 -3890.693,E2 -3890.693} C_VEL
LIN {X 0,Y 539.394,Z 283.856,A -85,B 0,C 180,E1 -3890.964,E2 -3890.964} C_VEL
LIN {X 0,Y 539.517,Z 273.118,A -85,B 0,C 180,E1 -3892.619,E2 -3892.619} C_VEL
LIN {X 0,Y 537.993,Z 266.097,A -85,B 0,C 180,E1 -3893.817,E2 -3893.817} C_VEL
LIN {X 0,Y 537.981,Z 266.095,A -85,B 0,C 180,E1 -3896.37,E2 -3896.37} C_VEL
LIN {X 0,Y 537.991,Z 266.1,A -85,B 0,C 180,E1 -3898.925,E2 -3898.925} C_VEL
LIN {X 0,Y 537.994,Z 266.094,A -85,B 0,C 180,E1 -3901.884,E2 -3901.884} C_VEL
LIN {X 0,Y 537.991,Z 266.097,A -85,B 0,C 180,E1 -3904.614,E2 -3904.614} C_VEL
LIN {X 0,Y 537.978,Z 266.094,A -85,B 0,C 180,E1 -3907.879,E2 -3907.879} C_VEL
LIN {X 0,Y 537.995,Z 266.098,A -85,B 0,C 180,E1 -3910.78,E2 -3910.78} C_VEL
LIN {X 0,Y 537.994,Z 266.089,A -85,B 0,C 180,E1 -3914.07,E2 -3914.07} C_VEL
LIN {X 0,Y 537.951,Z 266.096,A -85,B 0,C 180,E1 -3917.021,E2 -3917.021} C_VEL
LIN {X 0,Y 537.949,Z 266.097,A -85,B 0,C 180,E1 -3919.265,E2 -3919.265} C_VEL
LIN {X 0,Y 537.961,Z 266.095,A -85,B 0,C 180,E1 -3922.12,E2 -3922.12} C_VEL
LIN {X 0,Y 537.985,Z 266.091,A -85,B 0,C 180,E1 -3925.386,E2 -3925.386} C_VEL
LIN {X 0,Y 537.993,Z 266.093,A -85,B 0,C 180,E1 -3928.116,E2 -3928.116} C_VEL
LIN {X 0,Y 537.982,Z 266.094,A -85,B 0,C 180,E1 -3931.095,E2 -3931.095} C_VEL
LIN {X 0,Y 537.977,Z 266.092,A -85,B 0,C 180,E1 -3933.63,E2 -3933.63} C_VEL
LIN {X 0,Y 537.981,Z 266.095,A -85,B 0,C 180,E1 -3936.128,E2 -3936.128} C_VEL
LIN {X 0,Y 537.988,Z 266.1,A -85,B 0,C 180,E1 -3938.544,E2 -3938.544} C_VEL
LIN {X 0,Y 538.003,Z 266.089,A -85,B 0,C 180,E1 -3940.939,E2 -3940.939} C_VEL
LIN {X 0,Y 537.961,Z 266.094,A -85,B 0,C 180,E1 -3943.297,E2 -3943.297} C_VEL
LIN {X 0,Y 538.033,Z 266.084,A -85,B 0,C 180,E1 -3945.63,E2 -3945.63} C_VEL
LIN {X 0,Y 538.071,Z 266.084,A -85,B 0,C 180,E1 -3948.701,E2 -3948.701} C_VEL
LIN {X 0,Y 538.047,Z 266.083,A -85,B 0,C 180,E1 -3951.739,E2 -3951.739} C_VEL
LIN {X 0,Y 538.123,Z 266.075,A -85,B 0,C 180,E1 -3954.755,E2 -3954.755} C_VEL
LIN {X 0,Y 538.156,Z 266.072,A -85,B 0,C 180,E1 -3957.755,E2 -3957.755} C_VEL
LIN {X 0,Y 538.176,Z 266.066,A -85,B 0,C 180,E1 -3960.748,E2 -3960.748} C_VEL
LIN {X 0,Y 538.119,Z 266.075,A -85,B 0,C 180,E1 -3962.994,E2 -3962.994} C_VEL
LIN {X 0,Y 538.085,Z 266.085,A -85,B 0,C 180,E1 -3965.998,E2 -3965.998} C_VEL
LIN {X 0,Y 538.047,Z 266.083,A -85,B 0,C 180,E1 -3969.018,E2 -3969.018} C_VEL
LIN {X 0,Y 538.062,Z 266.09,A -85,B 0,C 180,E1 -3972.063,E2 -3972.063} C_VEL
LIN {X 0,Y 538.043,Z 266.082,A -85,B 0,C 180,E1 -3975.144,E2 -3975.144} C_VEL
LIN {X 0,Y 538.012,Z 266.092,A -85,B 0,C 180,E1 -3978.271,E2 -3978.271} C_VEL
LIN {X 0,Y 538.036,Z 266.086,A -85,B 0,C 180,E1 -3980.651,E2 -3980.651} C_VEL
LIN {X 0,Y 538,Z 266.092,A -85,B 0,C 180,E1 -3983.888,E2 -3983.888} C_VEL
LIN {X 0,Y 538.033,Z 266.085,A -85,B 0,C 180,E1 -3986.367,E2 -3986.367} C_VEL
LIN {X 0,Y 538.028,Z 266.086,A -85,B 0,C 180,E1 -3988.933,E2 -3988.933} C_VEL
LIN {X 0,Y 538.009,Z 266.09,A -85,B 0,C 180,E1 -3991.887,E2 -3991.887} C_VEL
LIN {X 0,Y 538.015,Z 266.088,A -85,B 0,C 180,E1 -3994.618,E2 -3994.618} C_VEL
LIN {X 0,Y 538.004,Z 266.088,A -85,B 0,C 180,E1 -3997.17,E2 -3997.17} C_VEL
LIN {X 0,Y 538.021,Z 266.095,A -85,B 0,C 180,E1 -3999.797,E2 -3999.797} C_VEL
LIN {X 0,Y 538.017,Z 266.088,A -85,B 0,C 180,E1 -4002.786,E2 -4002.786} C_VEL
LIN {X 0,Y 538.017,Z 266.091,A -85,B 0,C 180,E1 -4005.927,E2 -4005.927} C_VEL
LIN {X 0,Y 538.03,Z 266.086,A -85,B 0,C 180,E1 -4008.227,E2 -4008.227} C_VEL
LIN {X 0,Y 538.011,Z 266.092,A -85,B 0,C 180,E1 -4011.17,E2 -4011.17} C_VEL
LIN {X 0,Y 538.023,Z 266.09,A -85,B 0,C 180,E1 -4014.084,E2 -4014.084} C_VEL
LIN {X 0,Y 538.029,Z 266.087,A -85,B 0,C 180,E1 -4016.728,E2 -4016.728} C_VEL
LIN {X 0,Y 538.025,Z 266.094,A -85,B 0,C 180,E1 -4019.556,E2 -4019.556} C_VEL
LIN {X 0,Y 538.059,Z 266.175,A -85,B 0,C 180,E1 -4022.055,E2 -4022.055} C_VEL
LIN {X 0,Y 540.479,Z 276.823,A -85,B 0,C 180,E1 -4023.554,E2 -4023.554} C_VEL
LIN {X 0,Y 540.277,Z 291.399,A -85,B 0,C 180,E1 -4025.402,E2 -4025.402} C_VEL
LIN {X 0,Y 539.697,Z 314.042,A -85,B 0,C 180,E1 -4028.215,E2 -4028.215} C_VEL
LIN {X 0,Y 539.528,Z 321.082,A -85,B 0,C 180,E1 -4029.079,E2 -4029.079} C_VEL
LIN {X 0,Y 541.813,Z 332.998,A -85,B 0,C 180,E1 -4029.335,E2 -4029.335} C_VEL
LIN {X 0,Y 540.99,Z 487.946,A -85,B 0,C 180,E1 -4031.461,E2 -4031.461} C_VEL
LIN {X 0,Y 540.752,Z 503.342,A -85,B 0,C 180,E1 -4031.825,E2 -4031.825} C_VEL
LIN {X 0,Y 540.411,Z 518.719,A -85,B 0,C 180,E1 -4032.352,E2 -4032.352} C_VEL
LIN {X 0,Y 540.086,Z 532.525,A -85,B 0,C 180,E1 -4032.975,E2 -4032.975} C_VEL
LIN {X 0,Y 539.641,Z 546.057,A -85,B 0,C 180,E1 -4033.74,E2 -4033.74} C_VEL
LIN {X 0,Y 539.309,Z 559.185,A -85,B 0,C 180,E1 -4034.65,E2 -4034.65} C_VEL
LIN {X 0,Y 538.888,Z 571.246,A -85,B 0,C 180,E1 -4035.653,E2 -4035.653} C_VEL
LIN {X 0,Y 538.593,Z 582.749,A -85,B 0,C 180,E1 -4036.8,E2 -4036.8} C_VEL
LIN {X 0,Y 538.282,Z 592.39,A -85,B 0,C 180,E1 -4037.942,E2 -4037.942} C_VEL
LIN {X 0,Y 538.068,Z 601.855,A -85,B 0,C 180,E1 -4039.273,E2 -4039.273} C_VEL
LIN {X 0,Y 537.824,Z 609.736,A -85,B 0,C 180,E1 -4040.599,E2 -4040.599} C_VEL
LIN {X 0,Y 537.699,Z 617.09,A -85,B 0,C 180,E1 -4042.112,E2 -4042.112} C_VEL
LIN {X 0,Y 537.622,Z 622.406,A -85,B 0,C 180,E1 -4043.464,E2 -4043.464} C_VEL
LIN {X 0,Y 537.574,Z 626.387,A -85,B 0,C 180,E1 -4044.75,E2 -4044.75} C_VEL
LIN {X 0,Y 537.561,Z 629.888,A -85,B 0,C 180,E1 -4046.252,E2 -4046.252} C_VEL
LIN {X 0,Y 537.487,Z 632.19,A -85,B 0,C 180,E1 -4047.752,E2 -4047.752} C_VEL
LIN {X 0,Y 537.439,Z 633.348,A -85,B 0,C 180,E1 -4049.251,E2 -4049.251} C_VEL
LIN {X 0,Y 537.439,Z 633.347,A -85,B 0,C 180,E1 -4050.75,E2 -4050.75} C_VEL
LIN {X 0,Y 537.487,Z 632.185,A -85,B 0,C 180,E1 -4052.248,E2 -4052.248} C_VEL
LIN {X 0,Y 537.561,Z 629.882,A -85,B 0,C 180,E1 -4053.748,E2 -4053.748} C_VEL
LIN {X 0,Y 537.574,Z 626.385,A -85,B 0,C 180,E1 -4055.251,E2 -4055.251} C_VEL
LIN {X 0,Y 537.618,Z 621.608,A -85,B 0,C 180,E1 -4056.757,E2 -4056.757} C_VEL
LIN {X 0,Y 537.734,Z 615.418,A -85,B 0,C 180,E1 -4058.266,E2 -4058.266} C_VEL
LIN {X 0,Y 537.86,Z 607.64,A -85,B 0,C 180,E1 -4059.78,E2 -4059.78} C_VEL
LIN {X 0,Y 538.102,Z 599.363,A -85,B 0,C 180,E1 -4061.108,E2 -4061.108} C_VEL
LIN {X 0,Y 538.358,Z 589.388,A -85,B 0,C 180,E1 -4062.439,E2 -4062.439} C_VEL
LIN {X 0,Y 538.663,Z 579.179,A -85,B 0,C 180,E1 -4063.583,E2 -4063.583} C_VEL
LIN {X 0,Y 539.03,Z 566.939,A -85,B 0,C 180,E1 -4064.729,E2 -4064.729} C_VEL
LIN {X 0,Y 539.431,Z 554.667,A -85,B 0,C 180,E1 -4065.683,E2 -4065.683} C_VEL
LIN {X 0,Y 539.82,Z 541.272,A -85,B 0,C 180,E1 -4066.547,E2 -4066.547} C_VEL
LIN {X 0,Y 540.227,Z 526.521,A -85,B 0,C 180,E1 -4067.313,E2 -4067.313} C_VEL
LIN {X 0,Y 540.534,Z 512.259,A -85,B 0,C 180,E1 -4067.889,E2 -4067.889} C_VEL
LIN {X 0,Y 540.821,Z 497.389,A -85,B 0,C 180,E1 -4068.333,E2 -4068.333} C_VEL
LIN {X 0,Y 541.04,Z 482.472,A -85,B 0,C 180,E1 -4068.628,E2 -4068.628} C_VEL
LIN {X 0,Y 541.794,Z 332.652,A -85,B 0,C 180,E1 -4070.67,E2 -4070.67} C_VEL
LIN {X 0,Y 539.543,Z 320.989,A -85,B 0,C 180,E1 -4070.932,E2 -4070.932} C_VEL
LIN {X 0,Y 540.137,Z 296.655,A -85,B 0,C 180,E1 -4073.941,E2 -4073.941} C_VEL
LIN {X 0,Y 540.577,Z 278.44,A -85,B 0,C 180,E1 -4076.234,E2 -4076.234} C_VEL
LIN {X 0,Y 539.818,Z 273.54,A -85,B 0,C 180,E1 -4076.899,E2 -4076.899} C_VEL
LIN {X 0,Y 538.038,Z 266.092,A -85,B 0,C 180,E1 -4077.967,E2 -4077.967} C_VEL
LIN {X 0,Y 538.023,Z 266.093,A -85,B 0,C 180,E1 -4080.627,E2 -4080.627} C_VEL
LIN {X 0,Y 538.048,Z 266.086,A -85,B 0,C 180,E1 -4083.283,E2 -4083.283} C_VEL
LIN {X 0,Y 537.997,Z 266.093,A -85,B 0,C 180,E1 -4086.005,E2 -4086.005} C_VEL
LIN {X 0,Y 538.015,Z 266.089,A -85,B 0,C 180,E1 -4088.831,E2 -4088.831} C_VEL
LIN {X 0,Y 538.027,Z 266.087,A -85,B 0,C 180,E1 -4091.774,E2 -4091.774} C_VEL
LIN {X 0,Y 538.001,Z 266.092,A -85,B 0,C 180,E1 -4094.863,E2 -4094.863} C_VEL
LIN {X 0,Y 538.022,Z 266.086,A -85,B 0,C 180,E1 -4097.214,E2 -4097.214} C_VEL
LIN {X 0,Y 538.014,Z 266.095,A -85,B 0,C 180,E1 -4100.202,E2 -4100.202} C_VEL
LIN {X 0,Y 538.022,Z 266.087,A -85,B 0,C 180,E1 -4103.067,E2 -4103.067} C_VEL
LIN {X 0,Y 538.02,Z 266.089,A -85,B 0,C 180,E1 -4105.827,E2 -4105.827} C_VEL
LIN {X 0,Y 538.013,Z 266.092,A -85,B 0,C 180,E1 -4108.499,E2 -4108.499} C_VEL
LIN {X 0,Y 538.022,Z 266.085,A -85,B 0,C 180,E1 -4111.098,E2 -4111.098} C_VEL
LIN {X 0,Y 538.018,Z 266.088,A -85,B 0,C 180,E1 -4113.632,E2 -4113.632} C_VEL
LIN {X 0,Y 538.012,Z 266.096,A -85,B 0,C 180,E1 -4116.122,E2 -4116.122} C_VEL
LIN {X 0,Y 538.041,Z 266.085,A -85,B 0,C 180,E1 -4119.349,E2 -4119.349} C_VEL
LIN {X 0,Y 538.042,Z 266.088,A -85,B 0,C 180,E1 -4122.468,E2 -4122.468} C_VEL
LIN {X 0,Y 538.068,Z 266.083,A -85,B 0,C 180,E1 -4125.631,E2 -4125.631} C_VEL
LIN {X 0,Y 538.081,Z 266.078,A -85,B 0,C 180,E1 -4128.702,E2 -4128.702} C_VEL
LIN {X 0,Y 538.046,Z 266.09,A -85,B 0,C 180,E1 -4131.739,E2 -4131.739} C_VEL
LIN {X 0,Y 538.134,Z 266.073,A -85,B 0,C 180,E1 -4134.755,E2 -4134.755} C_VEL
LIN {X 0,Y 538.164,Z 266.075,A -85,B 0,C 180,E1 -4137.755,E2 -4137.755} C_VEL
LIN {X 0,Y 538.162,Z 266.075,A -85,B 0,C 180,E1 -4140,E2 -4140} C_VEL
LIN {X 0,Y 538.128,Z 266.073,A -85,B 0,C 180,E1 -4142.995,E2 -4142.995} C_VEL
LIN {X 0,Y 538.08,Z 266.084,A -85,B 0,C 180,E1 -4145.998,E2 -4145.998} C_VEL
LIN {X 0,Y 538.028,Z 266.087,A -85,B 0,C 180,E1 -4149.018,E2 -4149.018} C_VEL
LIN {X 0,Y 538.054,Z 266.087,A -85,B 0,C 180,E1 -4152.063,E2 -4152.063} C_VEL
LIN {X 0,Y 538.041,Z 266.084,A -85,B 0,C 180,E1 -4155.144,E2 -4155.144} C_VEL
LIN {X 0,Y 538,Z 266.089,A -85,B 0,C 180,E1 -4158.271,E2 -4158.271} C_VEL
LIN {X 0,Y 537.991,Z 266.091,A -85,B 0,C 180,E1 -4160.653,E2 -4160.653} C_VEL
LIN {X 0,Y 537.979,Z 266.093,A -85,B 0,C 180,E1 -4163.074,E2 -4163.074} C_VEL
LIN {X 0,Y 537.988,Z 266.096,A -85,B 0,C 180,E1 -4165.659,E2 -4165.659} C_VEL
LIN {X 0,Y 537.974,Z 266.089,A -85,B 0,C 180,E1 -4168.054,E2 -4168.054} C_VEL
LIN {X 0,Y 537.991,Z 266.09,A -85,B 0,C 180,E1 -4170.629,E2 -4170.629} C_VEL
LIN {X 0,Y 538.002,Z 266.096,A -85,B 0,C 180,E1 -4173.275,E2 -4173.275} C_VEL
LIN {X 0,Y 537.956,Z 266.095,A -85,B 0,C 180,E1 -4176.008,E2 -4176.008} C_VEL
LIN {X 0,Y 537.975,Z 266.094,A -85,B 0,C 180,E1 -4178.834,E2 -4178.834} C_VEL
LIN {X 0,Y 537.943,Z 266.096,A -85,B 0,C 180,E1 -4180.216,E2 -4180.216} C_VEL
LIN {X 0,Y 537.277,Z 266.182,A -85,B 0,C 180,E1 -4180.841,E2 -4180.841} C_VEL
LIN {X 0,Y 534.438,Z 266.542,A -85,B 0,C 180,E1 -4181.856,E2 -4181.856} C_VEL
LIN {X 0,Y 532.038,Z 266.844,A -85,B 0,C 180,E1 -4182.674,E2 -4182.674} C_VEL
LIN {X 0,Y 531.006,Z 266.969,A -85,B 0,C 180,E1 -4183.304,E2 -4183.304} C_VEL
LIN {X 0,Y 530.921,Z 266.977,A -85,B 0,C 180,E1 -4183.518,E2 -4183.518} C_VEL
LIN {X 0,Y 530.916,Z 266.975,A -85,B 0,C 180,E1 -4185.629,E2 -4185.629} C_VEL
LIN {X 0,Y 530.902,Z 266.974,A -85,B 0,C 180,E1 -4188.555,E2 -4188.555} C_VEL
LIN {X 0,Y 530.918,Z 266.976,A -85,B 0,C 180,E1 -4191.525,E2 -4191.525} C_VEL
LIN {X 0,Y 530.927,Z 266.972,A -85,B 0,C 180,E1 -4194.377,E2 -4194.377} C_VEL
LIN {X 0,Y 530.947,Z 266.977,A -85,B 0,C 180,E1 -4197.131,E2 -4197.131} C_VEL
LIN {X 0,Y 530.93,Z 266.973,A -85,B 0,C 180,E1 -4199.8,E2 -4199.8} C_VEL
LIN {X 0,Y 530.956,Z 266.97,A -85,B 0,C 180,E1 -4202.48,E2 -4202.48} C_VEL
LIN {X 0,Y 530.947,Z 266.975,A -85,B 0,C 180,E1 -4205.773,E2 -4205.773} C_VEL
LIN {X 0,Y 530.986,Z 267.193,A -85,B 0,C 180,E1 -4206.1,E2 -4206.1} C_VEL
LIN {X 0,Y 532.673,Z 275.497,A -85,B 0,C 180,E1 -4207.503,E2 -4207.503} C_VEL
LIN {X 0,Y 532.556,Z 284.192,A -85,B 0,C 180,E1 -4208.854,E2 -4208.854} C_VEL
LIN {X 0,Y 535.13,Z 295.449,A -85,B 0,C 180,E1 -4209.122,E2 -4209.122} C_VEL
LIN {X 0,Y 534.515,Z 415.687,A -85,B 0,C 180,E1 -4210.784,E2 -4210.784} C_VEL
LIN {X 0,Y 534.288,Z 449.774,A -85,B 0,C 180,E1 -4211.278,E2 -4211.278} C_VEL
LIN {X 0,Y 534.027,Z 465.374,A -85,B 0,C 180,E1 -4211.662,E2 -4211.662} C_VEL
LIN {X 0,Y 533.717,Z 479.847,A -85,B 0,C 180,E1 -4212.172,E2 -4212.172} C_VEL
LIN {X 0,Y 533.385,Z 492.524,A -85,B 0,C 180,E1 -4212.754,E2 -4212.754} C_VEL
LIN {X 0,Y 532.925,Z 506.12,A -85,B 0,C 180,E1 -4213.528,E2 -4213.528} C_VEL
LIN {X 0,Y 532.477,Z 519.58,A -85,B 0,C 180,E1 -4214.474,E2 -4214.474} C_VEL
LIN {X 0,Y 532.052,Z 531.248,A -85,B 0,C 180,E1 -4215.464,E2 -4215.464} C_VEL
LIN {X 0,Y 531.642,Z 542.699,A -85,B 0,C 180,E1 -4216.624,E2 -4216.624} C_VEL
LIN {X 0,Y 531.325,Z 552.331,A -85,B 0,C 180,E1 -4217.781,E2 -4217.781} C_VEL
LIN {X 0,Y 531.051,Z 561.766,A -85,B 0,C 180,E1 -4219.129,E2 -4219.129} C_VEL
LIN {X 0,Y 530.798,Z 569.622,A -85,B 0,C 180,E1 -4220.473,E2 -4220.473} C_VEL
LIN {X 0,Y 530.642,Z 576.952,A -85,B 0,C 180,E1 -4222.006,E2 -4222.006} C_VEL
LIN {X 0,Y 530.523,Z 582.629,A -85,B 0,C 180,E1 -4223.489,E2 -4223.489} C_VEL
LIN {X 0,Y 530.509,Z 586.26,A -85,B 0,C 180,E1 -4224.679,E2 -4224.679} C_VEL
LIN {X 0,Y 530.481,Z 589.795,A -85,B 0,C 180,E1 -4226.201,E2 -4226.201} C_VEL
LIN {X 0,Y 530.409,Z 592.137,A -85,B 0,C 180,E1 -4227.721,E2 -4227.721} C_VEL
LIN {X 0,Y 530.34,Z 593.337,A -85,B 0,C 180,E1 -4229.24,E2 -4229.24} C_VEL
LIN {X 0,Y 530.341,Z 593.357,A -85,B 0,C 180,E1 -4230.759,E2 -4230.759} C_VEL
LIN {X 0,Y 530.409,Z 592.236,A -85,B 0,C 180,E1 -4232.278,E2 -4232.278} C_VEL
LIN {X 0,Y 530.482,Z 589.973,A -85,B 0,C 180,E1 -4233.798,E2 -4233.798} C_VEL
LIN {X 0,Y 530.507,Z 586.512,A -85,B 0,C 180,E1 -4235.321,E2 -4235.321} C_VEL
LIN {X 0,Y 530.55,Z 581.778,A -85,B 0,C 180,E1 -4236.847,E2 -4236.847} C_VEL
LIN {X 0,Y 530.665,Z 575.706,A -85,B 0,C 180,E1 -4238.376,E2 -4238.376} C_VEL
LIN {X 0,Y 530.819,Z 568.059,A -85,B 0,C 180,E1 -4239.911,E2 -4239.911} C_VEL
LIN {X 0,Y 531.06,Z 559.899,A -85,B 0,C 180,E1 -4241.256,E2 -4241.256} C_VEL
LIN {X 0,Y 531.398,Z 550.069,A -85,B 0,C 180,E1 -4242.604,E2 -4242.604} C_VEL
LIN {X 0,Y 531.739,Z 539.986,A -85,B 0,C 180,E1 -4243.763,E2 -4243.763} C_VEL
LIN {X 0,Y 532.135,Z 527.98,A -85,B 0,C 180,E1 -4244.924,E2 -4244.924} C_VEL
LIN {X 0,Y 532.612,Z 515.924,A -85,B 0,C 180,E1 -4245.891,E2 -4245.891} C_VEL
LIN {X 0,Y 533.061,Z 502.852,A -85,B 0,C 180,E1 -4246.762,E2 -4246.762} C_VEL
LIN {X 0,Y 533.439,Z 490.39,A -85,B 0,C 180,E1 -4247.441,E2 -4247.441} C_VEL
LIN {X 0,Y 533.833,Z 475.809,A -85,B 0,C 180,E1 -4248.071,E2 -4248.071} C_VEL
LIN {X 0,Y 534.123,Z 460.185,A -85,B 0,C 180,E1 -4248.571,E2 -4248.571} C_VEL
LIN {X 0,Y 534.364,Z 444.735,A -85,B 0,C 180,E1 -4248.897,E2 -4248.897} C_VEL
LIN {X 0,Y 535.239,Z 296.689,A -85,B 0,C 180,E1 -4250.946,E2 -4250.946} C_VEL
LIN {X 0,Y 532.546,Z 284.054,A -85,B 0,C 180,E1 -4251.255,E2 -4251.255} C_VEL
LIN {X 0,Y 532.71,Z 275.682,A -85,B 0,C 180,E1 -4252.556,E2 -4252.556} C_VEL
LIN {X 0,Y 530.952,Z 266.974,A -85,B 0,C 180,E1 -4254.031,E2 -4254.031} C_VEL
LIN {X 0,Y 530.944,Z 266.976,A -85,B 0,C 180,E1 -4256.747,E2 -4256.747} C_VEL
LIN {X 0,Y 530.953,Z 266.975,A -85,B 0,C 180,E1 -4259.324,E2 -4259.324} C_VEL
LIN {X 0,Y 530.95,Z 266.972,A -85,B 0,C 180,E1 -4262.097,E2 -4262.097} C_VEL
LIN {X 0,Y 530.953,Z 266.978,A -85,B 0,C 180,E1 -4264.848,E2 -4264.848} C_VEL
LIN {X 0,Y 530.93,Z 266.973,A -85,B 0,C 180,E1 -4267.51,E2 -4267.51} C_VEL
LIN {X 0,Y 530.943,Z 266.973,A -85,B 0,C 180,E1 -4270.436,E2 -4270.436} C_VEL
LIN {X 0,Y 530.918,Z 266.971,A -85,B 0,C 180,E1 -4273.499,E2 -4273.499} C_VEL
LIN {X 0,Y 530.959,Z 266.967,A -85,B 0,C 180,E1 -4275.624,E2 -4275.624} C_VEL
LIN {X 0,Y 530.905,Z 266.974,A -85,B 0,C 180,E1 -4278.556,E2 -4278.556} C_VEL
LIN {X 0,Y 530.919,Z 266.971,A -85,B 0,C 180,E1 -4281.526,E2 -4281.526} C_VEL
LIN {X 0,Y 530.921,Z 266.968,A -85,B 0,C 180,E1 -4284.377,E2 -4284.377} C_VEL
LIN {X 0,Y 530.943,Z 266.971,A -85,B 0,C 180,E1 -4287.132,E2 -4287.132} C_VEL
LIN {X 0,Y 530.927,Z 266.97,A -85,B 0,C 180,E1 -4289.8,E2 -4289.8} C_VEL
LIN {X 0,Y 530.952,Z 266.974,A -85,B 0,C 180,E1 -4292.48,E2 -4292.48} C_VEL
LIN {X 0,Y 530.941,Z 266.972,A -85,B 0,C 180,E1 -4294.939,E2 -4294.939} C_VEL
LIN {X 0,Y 530.946,Z 266.973,A -85,B 0,C 180,E1 -4298.245,E2 -4298.245} C_VEL
LIN {X 0,Y 530.957,Z 266.97,A -85,B 0,C 180,E1 -4300.676,E2 -4300.676} C_VEL
LIN {X 0,Y 530.926,Z 266.972,A -85,B 0,C 180,E1 -4303.069,E2 -4303.069} C_VEL
LIN {X 0,Y 530.995,Z 266.96,A -85,B 0,C 180,E1 -4305.435,E2 -4305.435} C_VEL
LIN {X 0,Y 531.03,Z 266.964,A -85,B 0,C 180,E1 -4308.549,E2 -4308.549} C_VEL
LIN {X 0,Y 530.993,Z 266.961,A -85,B 0,C 180,E1 -4311.628,E2 -4311.628} C_VEL
LIN {X 0,Y 531.083,Z 266.952,A -85,B 0,C 180,E1 -4314.685,E2 -4314.685} C_VEL
LIN {X 0,Y 531.129,Z 266.947,A -85,B 0,C 180,E1 -4317.725,E2 -4317.725} C_VEL
LIN {X 0,Y 531.147,Z 266.941,A -85,B 0,C 180,E1 -4320.758,E2 -4320.758} C_VEL
LIN {X 0,Y 531.085,Z 266.951,A -85,B 0,C 180,E1 -4323.034,E2 -4323.034} C_VEL
LIN {X 0,Y 531.044,Z 266.961,A -85,B 0,C 180,E1 -4326.077,E2 -4326.077} C_VEL
LIN {X 0,Y 531.01,Z 266.96,A -85,B 0,C 180,E1 -4329.138,E2 -4329.138} C_VEL
LIN {X 0,Y 531.048,Z 266.957,A -85,B 0,C 180,E1 -4331.67,E2 -4331.67} C_VEL
LIN {X 0,Y 531.03,Z 266.955,A -85,B 0,C 180,E1 -4334.956,E2 -4334.956} C_VEL
LIN {X 0,Y 530.979,Z 266.97,A -85,B 0,C 180,E1 -4337.724,E2 -4337.724} C_VEL
LIN {X 0,Y 531.024,Z 266.965,A -85,B 0,C 180,E1 -4340.127,E2 -4340.127} C_VEL
LIN {X 0,Y 530.943,Z 266.969,A -85,B 0,C 180,E1 -4342.573,E2 -4342.573} C_VEL
LIN {X 0,Y 530.987,Z 266.956,A -85,B 0,C 180,E1 -4345.058,E2 -4345.058} C_VEL
LIN {X 0,Y 530.968,Z 266.968,A -85,B 0,C 180,E1 -4347.598,E2 -4347.598} C_VEL
LIN {X 0,Y 530.967,Z 266.966,A -85,B 0,C 180,E1 -4350.197,E2 -4350.197} C_VEL
LIN {X 0,Y 530.966,Z 266.962,A -85,B 0,C 180,E1 -4352.867,E2 -4352.867} C_VEL
LIN {X 0,Y 530.96,Z 266.974,A -85,B 0,C 180,E1 -4355.62,E2 -4355.62} C_VEL
LIN {X 0,Y 530.963,Z 266.965,A -85,B 0,C 180,E1 -4358.653,E2 -4358.653} C_VEL
LIN {X 0,Y 530.992,Z 266.968,A -85,B 0,C 180,E1 -4361.436,E2 -4361.436} C_VEL
LIN {X 0,Y 530.971,Z 266.965,A -85,B 0,C 180,E1 -4364.549,E2 -4364.549} C_VEL
LIN {X 0,Y 530.981,Z 266.968,A -85,B 0,C 180,E1 -4367.834,E2 -4367.834} C_VEL
LIN {X 0,Y 530.984,Z 266.964,A -85,B 0,C 180,E1 -4370.557,E2 -4370.557} C_VEL
LIN {X 0,Y 530.965,Z 266.975,A -85,B 0,C 180,E1 -4373.443,E2 -4373.443} C_VEL
LIN {X 0,Y 530.998,Z 266.963,A -85,B 0,C 180,E1 -4376.494,E2 -4376.494} C_VEL
LIN {X 0,Y 530.973,Z 266.972,A -85,B 0,C 180,E1 -4379.355,E2 -4379.355} C_VEL
LIN {X 0,Y 531.024,Z 267.147,A -85,B 0,C 180,E1 -4381.816,E2 -4381.816} C_VEL
LIN {X 0,Y 533.589,Z 278.184,A -85,B 0,C 180,E1 -4383.396,E2 -4383.396} C_VEL
LIN {X 0,Y 533.61,Z 284.669,A -85,B 0,C 180,E1 -4384.238,E2 -4384.238} C_VEL
LIN {X 0,Y 533.059,Z 305.678,A -85,B 0,C 180,E1 -4386.907,E2 -4386.907} C_VEL
LIN {X 0,Y 532.644,Z 320.812,A -85,B 0,C 180,E1 -4388.796,E2 -4388.796} C_VEL
LIN {X 0,Y 535.166,Z 333.988,A -85,B 0,C 180,E1 -4389.084,E2 -4389.084} C_VEL
LIN {X 0,Y 534.25,Z 487.704,A -85,B 0,C 180,E1 -4391.219,E2 -4391.219} C_VEL
LIN {X 0,Y 533.996,Z 503.071,A -85,B 0,C 180,E1 -4391.587,E2 -4391.587} C_VEL
LIN {X 0,Y 533.634,Z 518.448,A -85,B 0,C 180,E1 -4392.12,E2 -4392.12} C_VEL
LIN {X 0,Y 533.25,Z 532.252,A -85,B 0,C 180,E1 -4392.75,E2 -4392.75} C_VEL
LIN {X 0,Y 532.779,Z 545.784,A -85,B 0,C 180,E1 -4393.524,E2 -4393.524} C_VEL
LIN {X 0,Y 532.412,Z 558.437,A -85,B 0,C 180,E1 -4394.411,E2 -4394.411} C_VEL
LIN {X 0,Y 531.954,Z 570.973,A -85,B 0,C 180,E1 -4395.462,E2 -4395.462} C_VEL
LIN {X 0,Y 531.575,Z 582.518,A -85,B 0,C 180,E1 -4396.623,E2 -4396.623} C_VEL
LIN {X 0,Y 531.254,Z 592.239,A -85,B 0,C 180,E1 -4397.78,E2 -4397.78} C_VEL
LIN {X 0,Y 531.051,Z 601.792,A -85,B 0,C 180,E1 -4399.13,E2 -4399.13} C_VEL
LIN {X 0,Y 530.764,Z 609.735,A -85,B 0,C 180,E1 -4400.473,E2 -4400.473} C_VEL
LIN {X 0,Y 530.639,Z 617.09,A -85,B 0,C 180,E1 -4402.007,E2 -4402.007} C_VEL
LIN {X 0,Y 530.542,Z 622.708,A -85,B 0,C 180,E1 -4403.469,E2 -4403.469} C_VEL
LIN {X 0,Y 530.508,Z 626.386,A -85,B 0,C 180,E1 -4404.679,E2 -4404.679} C_VEL
LIN {X 0,Y 530.48,Z 629.887,A -85,B 0,C 180,E1 -4406.202,E2 -4406.202} C_VEL
LIN {X 0,Y 530.408,Z 632.189,A -85,B 0,C 180,E1 -4407.722,E2 -4407.722} C_VEL
LIN {X 0,Y 530.341,Z 633.347,A -85,B 0,C 180,E1 -4409.241,E2 -4409.241} C_VEL
LIN {X 0,Y 530.341,Z 633.346,A -85,B 0,C 180,E1 -4410.76,E2 -4410.76} C_VEL
LIN {X 0,Y 530.408,Z 632.185,A -85,B 0,C 180,E1 -4412.279,E2 -4412.279} C_VEL
LIN {X 0,Y 530.48,Z 629.881,A -85,B 0,C 180,E1 -4413.799,E2 -4413.799} C_VEL
LIN {X 0,Y 530.508,Z 626.385,A -85,B 0,C 180,E1 -4415.321,E2 -4415.321} C_VEL
LIN {X 0,Y 530.55,Z 621.608,A -85,B 0,C 180,E1 -4416.847,E2 -4416.847} C_VEL
LIN {X 0,Y 530.665,Z 615.417,A -85,B 0,C 180,E1 -4418.377,E2 -4418.377} C_VEL
LIN {X 0,Y 530.809,Z 607.628,A -85,B 0,C 180,E1 -4419.912,E2 -4419.912} C_VEL
LIN {X 0,Y 531.057,Z 599.274,A -85,B 0,C 180,E1 -4421.257,E2 -4421.257} C_VEL
LIN {X 0,Y 531.348,Z 589.21,A -85,B 0,C 180,E1 -4422.606,E2 -4422.606} C_VEL
LIN {X 0,Y 531.684,Z 578.92,A -85,B 0,C 180,E1 -4423.765,E2 -4423.765} C_VEL
LIN {X 0,Y 532.104,Z 566.666,A -85,B 0,C 180,E1 -4424.925,E2 -4424.925} C_VEL
LIN {X 0,Y 532.564,Z 553.167,A -85,B 0,C 180,E1 -4425.982,E2 -4425.982} C_VEL
LIN {X 0,Y 533.052,Z 539.37,A -85,B 0,C 180,E1 -4426.862,E2 -4426.862} C_VEL
LIN {X 0,Y 533.455,Z 525.225,A -85,B 0,C 180,E1 -4427.59,E2 -4427.59} C_VEL
LIN {X 0,Y 533.794,Z 510.675,A -85,B 0,C 180,E1 -4428.173,E2 -4428.173} C_VEL
LIN {X 0,Y 534.127,Z 495.137,A -85,B 0,C 180,E1 -4428.624,E2 -4428.624} C_VEL
LIN {X 0,Y 534.33,Z 480.287,A -85,B 0,C 180,E1 -4428.903,E2 -4428.903} C_VEL
LIN {X 0,Y 535.146,Z 333.681,A -85,B 0,C 180,E1 -4430.921,E2 -4430.921} C_VEL
LIN {X 0,Y 532.653,Z 320.802,A -85,B 0,C 180,E1 -4431.205,E2 -4431.205} C_VEL
LIN {X 0,Y 533.271,Z 297.606,A -85,B 0,C 180,E1 -4434.114,E2 -4434.114} C_VEL
LIN {X 0,Y 533.725,Z 279.399,A -85,B 0,C 180,E1 -4436.439,E2 -4436.439} C_VEL
LIN {X 0,Y 531.808,Z 270.524,A -85,B 0,C 180,E1 -4437.696,E2 -4437.696} C_VEL
LIN {X 0,Y 530.984,Z 266.972,A -85,B 0,C 180,E1 -4438.241,E2 -4438.241} C_VEL
LIN {X 0,Y 530.959,Z 266.97,A -85,B 0,C 180,E1 -4441.08,E2 -4441.08} C_VEL
LIN {X 0,Y 530.989,Z 266.965,A -85,B 0,C 180,E1 -4443.773,E2 -4443.773} C_VEL
LIN {X 0,Y 530.958,Z 266.975,A -85,B 0,C 180,E1 -4446.559,E2 -4446.559} C_VEL
LIN {X 0,Y 530.988,Z 266.96,A -85,B 0,C 180,E1 -4449.444,E2 -4449.444} C_VEL
LIN {X 0,Y 530.961,Z 266.975,A -85,B 0,C 180,E1 -4452.459,E2 -4452.459} C_VEL
LIN {X 0,Y 530.978,Z 266.965,A -85,B 0,C 180,E1 -4455.623,E2 -4455.623} C_VEL
LIN {X 0,Y 530.996,Z 266.968,A -85,B 0,C 180,E1 -4458.565,E2 -4458.565} C_VEL
LIN {X 0,Y 530.957,Z 266.967,A -85,B 0,C 180,E1 -4461.529,E2 -4461.529} C_VEL
LIN {X 0,Y 530.952,Z 266.973,A -85,B 0,C 180,E1 -4464.38,E2 -4464.38} C_VEL
LIN {X 0,Y 530.971,Z 266.963,A -85,B 0,C 180,E1 -4467.134,E2 -4467.134} C_VEL
LIN {X 0,Y 530.973,Z 266.967,A -85,B 0,C 180,E1 -4469.803,E2 -4469.803} C_VEL
LIN {X 0,Y 530.97,Z 266.968,A -85,B 0,C 180,E1 -4472.478,E2 -4472.478} C_VEL
LIN {X 0,Y 530.983,Z 266.963,A -85,B 0,C 180,E1 -4474.941,E2 -4474.941} C_VEL
LIN {X 0,Y 530.976,Z 266.972,A -85,B 0,C 180,E1 -4478.247,E2 -4478.247} C_VEL
LIN {X 0,Y 530.987,Z 266.963,A -85,B 0,C 180,E1 -4480.677,E2 -4480.677} C_VEL
LIN {X 0,Y 530.968,Z 266.965,A -85,B 0,C 180,E1 -4483.07,E2 -4483.07} C_VEL
LIN {X 0,Y 531.024,Z 266.958,A -85,B 0,C 180,E1 -4485.436,E2 -4485.436} C_VEL
LIN {X 0,Y 531.04,Z 266.956,A -85,B 0,C 180,E1 -4488.55,E2 -4488.55} C_VEL
LIN {X 0,Y 530.996,Z 266.967,A -85,B 0,C 180,E1 -4491.629,E2 -4491.629} C_VEL
LIN {X 0,Y 531.095,Z 266.95,A -85,B 0,C 180,E1 -4494.685,E2 -4494.685} C_VEL
LIN {X 0,Y 531.137,Z 266.95,A -85,B 0,C 180,E1 -4497.725,E2 -4497.725} C_VEL
LIN {X 0,Y 531.131,Z 266.951,A -85,B 0,C 180,E1 -4500,E2 -4500} C_VEL
LIN {X 0,Y 531.096,Z 266.949,A -85,B 0,C 180,E1 -4503.034,E2 -4503.034} C_VEL
LIN {X 0,Y 531.039,Z 266.96,A -85,B 0,C 180,E1 -4506.078,E2 -4506.078} C_VEL
LIN {X 0,Y 530.994,Z 266.964,A -85,B 0,C 180,E1 -4509.139,E2 -4509.139} C_VEL
LIN {X 0,Y 531.053,Z 266.962,A -85,B 0,C 180,E1 -4511.669,E2 -4511.669} C_VEL
LIN {X 0,Y 531.023,Z 266.957,A -85,B 0,C 180,E1 -4514.95,E2 -4514.95} C_VEL
LIN {X 0,Y 530.975,Z 266.97,A -85,B 0,C 180,E1 -4517.724,E2 -4517.724} C_VEL
LIN {X 0,Y 530.976,Z 266.967,A -85,B 0,C 180,E1 -4520.129,E2 -4520.129} C_VEL
LIN {X 0,Y 530.92,Z 266.969,A -85,B 0,C 180,E1 -4522.575,E2 -4522.575} C_VEL
LIN {X 0,Y 530.942,Z 266.971,A -85,B 0,C 180,E1 -4525.061,E2 -4525.061} C_VEL
LIN {X 0,Y 530.954,Z 266.967,A -85,B 0,C 180,E1 -4527.599,E2 -4527.599} C_VEL
LIN {X 0,Y 530.945,Z 266.968,A -85,B 0,C 180,E1 -4530.639,E2 -4530.639} C_VEL
LIN {X 0,Y 530.949,Z 266.976,A -85,B 0,C 180,E1 -4533.496,E2 -4533.496} C_VEL
LIN {X 0,Y 530.902,Z 266.973,A -85,B 0,C 180,E1 -4536.146,E2 -4536.146} C_VEL
LIN {X 0,Y 530.933,Z 266.97,A -85,B 0,C 180,E1 -4538.648,E2 -4538.648} C_VEL
LIN {X 0,Y 530.91,Z 266.98,A -85,B 0,C 180,E1 -4541.444,E2 -4541.444} C_VEL
LIN {X 0,Y 530.921,Z 266.977,A -85,B 0,C 180,E1 -4543.518,E2 -4543.518} C_VEL
LIN {X 0,Y 530.255,Z 267.056,A -85,B 0,C 180,E1 -4544.152,E2 -4544.152} C_VEL
LIN {X 0,Y 527.41,Z 267.416,A -85,B 0,C 180,E1 -4545.18,E2 -4545.18} C_VEL
LIN {X 0,Y 524.998,Z 267.715,A -85,B 0,C 180,E1 -4546.008,E2 -4546.008} C_VEL
LIN {X 0,Y 523.949,Z 267.843,A -85,B 0,C 180,E1 -4546.648,E2 -4546.648} C_VEL
LIN {X 0,Y 523.857,Z 267.853,A -85,B 0,C 180,E1 -4546.864,E2 -4546.864} C_VEL
LIN {X 0,Y 523.865,Z 267.851,A -85,B 0,C 180,E1 -4549.912,E2 -4549.912} C_VEL
LIN {X 0,Y 523.849,Z 267.856,A -85,B 0,C 180,E1 -4552.862,E2 -4552.862} C_VEL
LIN {X 0,Y 523.903,Z 267.847,A -85,B 0,C 180,E1 -4555.707,E2 -4555.707} C_VEL
LIN {X 0,Y 523.907,Z 267.846,A -85,B 0,C 180,E1 -4558.454,E2 -4558.454} C_VEL
LIN {X 0,Y 523.873,Z 267.857,A -85,B 0,C 180,E1 -4561.121,E2 -4561.121} C_VEL
LIN {X 0,Y 523.879,Z 267.852,A -85,B 0,C 180,E1 -4564.004,E2 -4564.004} C_VEL
LIN {X 0,Y 523.948,Z 268.02,A -85,B 0,C 180,E1 -4565.853,E2 -4565.853} C_VEL
LIN {X 0,Y 525.84,Z 277.215,A -85,B 0,C 180,E1 -4567.43,E2 -4567.43} C_VEL
LIN {X 0,Y 525.697,Z 284.398,A -85,B 0,C 180,E1 -4568.556,E2 -4568.556} C_VEL
LIN {X 0,Y 528.577,Z 297.02,A -85,B 0,C 180,E1 -4568.868,E2 -4568.868} C_VEL
LIN {X 0,Y 527.633,Z 447.258,A -85,B 0,C 180,E1 -4570.981,E2 -4570.981} C_VEL
LIN {X 0,Y 527.411,Z 461.813,A -85,B 0,C 180,E1 -4571.311,E2 -4571.311} C_VEL
LIN {X 0,Y 527.035,Z 476.331,A -85,B 0,C 180,E1 -4571.787,E2 -4571.787} C_VEL
LIN {X 0,Y 526.658,Z 490.831,A -85,B 0,C 180,E1 -4572.427,E2 -4572.427} C_VEL
LIN {X 0,Y 526.185,Z 504.826,A -85,B 0,C 180,E1 -4573.211,E2 -4573.211} C_VEL
LIN {X 0,Y 525.676,Z 517.611,A -85,B 0,C 180,E1 -4574.093,E2 -4574.093} C_VEL
LIN {X 0,Y 525.212,Z 530.464,A -85,B 0,C 180,E1 -4575.172,E2 -4575.172} C_VEL
LIN {X 0,Y 524.762,Z 541.209,A -85,B 0,C 180,E1 -4576.248,E2 -4576.248} C_VEL
LIN {X 0,Y 524.383,Z 551.136,A -85,B 0,C 180,E1 -4577.42,E2 -4577.42} C_VEL
LIN {X 0,Y 524.063,Z 560.825,A -85,B 0,C 180,E1 -4578.787,E2 -4578.787} C_VEL
LIN {X 0,Y 523.797,Z 568.897,A -85,B 0,C 180,E1 -4580.149,E2 -4580.149} C_VEL
LIN {X 0,Y 523.615,Z 575.553,A -85,B 0,C 180,E1 -4581.509,E2 -4581.509} C_VEL
LIN {X 0,Y 523.483,Z 581.721,A -85,B 0,C 180,E1 -4583.06,E2 -4583.06} C_VEL
LIN {X 0,Y 523.442,Z 586.484,A -85,B 0,C 180,E1 -4584.607,E2 -4584.607} C_VEL
LIN {X 0,Y 523.402,Z 589.976,A -85,B 0,C 180,E1 -4586.15,E2 -4586.15} C_VEL
LIN {X 0,Y 523.332,Z 592.291,A -85,B 0,C 180,E1 -4587.691,E2 -4587.691} C_VEL
LIN {X 0,Y 523.246,Z 593.479,A -85,B 0,C 180,E1 -4589.23,E2 -4589.23} C_VEL
LIN {X 0,Y 523.247,Z 593.499,A -85,B 0,C 180,E1 -4590.769,E2 -4590.769} C_VEL
LIN {X 0,Y 523.333,Z 592.388,A -85,B 0,C 180,E1 -4592.309,E2 -4592.309} C_VEL
LIN {X 0,Y 523.403,Z 590.15,A -85,B 0,C 180,E1 -4593.849,E2 -4593.849} C_VEL
LIN {X 0,Y 523.439,Z 586.73,A -85,B 0,C 180,E1 -4595.393,E2 -4595.393} C_VEL
LIN {X 0,Y 523.481,Z 582.047,A -85,B 0,C 180,E1 -4596.94,E2 -4596.94} C_VEL
LIN {X 0,Y 523.612,Z 575.975,A -85,B 0,C 180,E1 -4598.49,E2 -4598.49} C_VEL
LIN {X 0,Y 523.795,Z 568.327,A -85,B 0,C 180,E1 -4600.045,E2 -4600.045} C_VEL
LIN {X 0,Y 524.06,Z 560.167,A -85,B 0,C 180,E1 -4601.408,E2 -4601.408} C_VEL
LIN {X 0,Y 524.432,Z 550.337,A -85,B 0,C 180,E1 -4602.774,E2 -4602.774} C_VEL
LIN {X 0,Y 524.804,Z 540.253,A -85,B 0,C 180,E1 -4603.948,E2 -4603.948} C_VEL
LIN {X 0,Y 525.256,Z 528.245,A -85,B 0,C 180,E1 -4605.124,E2 -4605.124} C_VEL
LIN {X 0,Y 525.826,Z 515.045,A -85,B 0,C 180,E1 -4606.191,E2 -4606.191} C_VEL
LIN {X 0,Y 526.345,Z 501.538,A -85,B 0,C 180,E1 -4607.082,E2 -4607.082} C_VEL
LIN {X 0,Y 526.795,Z 486.653,A -85,B 0,C 180,E1 -4607.869,E2 -4607.869} C_VEL
LIN {X 0,Y 527.198,Z 472.156,A -85,B 0,C 180,E1 -4608.458,E2 -4608.458} C_VEL
LIN {X 0,Y 527.478,Z 456.638,A -85,B 0,C 180,E1 -4608.917,E2 -4608.917} C_VEL
LIN {X 0,Y 527.691,Z 440.928,A -85,B 0,C 180,E1 -4609.212,E2 -4609.212} C_VEL
LIN {X 0,Y 528.607,Z 297.139,A -85,B 0,C 180,E1 -4611.219,E2 -4611.219} C_VEL
LIN {X 0,Y 525.706,Z 284.38,A -85,B 0,C 180,E1 -4611.536,E2 -4611.536} C_VEL
LIN {X 0,Y 525.77,Z 276.79,A -85,B 0,C 180,E1 -4612.731,E2 -4612.731} C_VEL
LIN {X 0,Y 523.919,Z 267.851,A -85,B 0,C 180,E1 -4614.281,E2 -4614.281} C_VEL
LIN {X 0,Y 523.893,Z 267.856,A -85,B 0,C 180,E1 -4617.136,E2 -4617.136} C_VEL
LIN {X 0,Y 523.882,Z 267.852,A -85,B 0,C 180,E1 -4619.759,E2 -4619.759} C_VEL
LIN {X 0,Y 523.894,Z 267.853,A -85,B 0,C 180,E1 -4622.452,E2 -4622.452} C_VEL
LIN {X 0,Y 523.906,Z 267.85,A -85,B 0,C 180,E1 -4625.227,E2 -4625.227} C_VEL
LIN {X 0,Y 523.898,Z 267.848,A -85,B 0,C 180,E1 -4628.103,E2 -4628.103} C_VEL
LIN {X 0,Y 523.912,Z 267.847,A -85,B 0,C 180,E1 -4631.304,E2 -4631.304} C_VEL
LIN {X 0,Y 523.928,Z 267.848,A -85,B 0,C 180,E1 -4634.688,E2 -4634.688} C_VEL
LIN {X 0,Y 523.883,Z 267.842,A -85,B 0,C 180,E1 -4637.874,E2 -4637.874} C_VEL
LIN {X 0,Y 523.887,Z 267.851,A -85,B 0,C 180,E1 -4641.084,E2 -4641.084} C_VEL
LIN {X 0,Y 523.85,Z 267.844,A -85,B 0,C 180,E1 -4643.821,E2 -4643.821} C_VEL
LIN {X 0,Y 523.894,Z 267.855,A -85,B 0,C 180,E1 -4646.632,E2 -4646.632} C_VEL
LIN {X 0,Y 523.904,Z 267.845,A -85,B 0,C 180,E1 -4649.352,E2 -4649.352} C_VEL
LIN {X 0,Y 523.909,Z 267.85,A -85,B 0,C 180,E1 -4652.295,E2 -4652.295} C_VEL
LIN {X 0,Y 523.897,Z 267.846,A -85,B 0,C 180,E1 -4655.426,E2 -4655.426} C_VEL
LIN {X 0,Y 523.918,Z 267.844,A -85,B 0,C 180,E1 -4657.938,E2 -4657.938} C_VEL
LIN {X 0,Y 523.935,Z 267.848,A -85,B 0,C 180,E1 -4660.406,E2 -4660.406} C_VEL
LIN {X 0,Y 523.893,Z 267.85,A -85,B 0,C 180,E1 -4662.835,E2 -4662.835} C_VEL
LIN {X 0,Y 523.958,Z 267.837,A -85,B 0,C 180,E1 -4665.235,E2 -4665.235} C_VEL
LIN {X 0,Y 524.013,Z 267.84,A -85,B 0,C 180,E1 -4668.394,E2 -4668.394} C_VEL
LIN {X 0,Y 523.953,Z 267.837,A -85,B 0,C 180,E1 -4671.515,E2 -4671.515} C_VEL
LIN {X 0,Y 524.029,Z 267.832,A -85,B 0,C 180,E1 -4674.613,E2 -4674.613} C_VEL
LIN {X 0,Y 524.102,Z 267.822,A -85,B 0,C 180,E1 -4677.694,E2 -4677.694} C_VEL
LIN {X 0,Y 524.117,Z 267.817,A -85,B 0,C 180,E1 -4680.768,E2 -4680.768} C_VEL
LIN {X 0,Y 524.026,Z 267.83,A -85,B 0,C 180,E1 -4683.075,E2 -4683.075} C_VEL
LIN {X 0,Y 524.006,Z 267.838,A -85,B 0,C 180,E1 -4686.159,E2 -4686.159} C_VEL
LIN {X 0,Y 523.98,Z 267.836,A -85,B 0,C 180,E1 -4689.262,E2 -4689.262} C_VEL
LIN {X 0,Y 523.998,Z 267.836,A -85,B 0,C 180,E1 -4691.737,E2 -4691.737} C_VEL
LIN {X 0,Y 523.993,Z 267.832,A -85,B 0,C 180,E1 -4695.052,E2 -4695.052} C_VEL
LIN {X 0,Y 523.943,Z 267.849,A -85,B 0,C 180,E1 -4697.97,E2 -4697.97} C_VEL
LIN {X 0,Y 523.971,Z 267.84,A -85,B 0,C 180,E1 -4700.41,E2 -4700.41} C_VEL
LIN {X 0,Y 523.909,Z 267.844,A -85,B 0,C 180,E1 -4702.894,E2 -4702.894} C_VEL
LIN {X 0,Y 523.928,Z 267.837,A -85,B 0,C 180,E1 -4705.42,E2 -4705.42} C_VEL
LIN {X 0,Y 523.916,Z 267.851,A -85,B 0,C 180,E1 -4708.002,E2 -4708.002} C_VEL
LIN {X 0,Y 523.943,Z 267.837,A -85,B 0,C 180,E1 -4710.855,E2 -4710.855} C_VEL
LIN {X 0,Y 523.958,Z 267.844,A -85,B 0,C 180,E1 -4713.735,E2 -4713.735} C_VEL
LIN {X 0,Y 523.906,Z 267.843,A -85,B 0,C 180,E1 -4716.402,E2 -4716.402} C_VEL
LIN {X 0,Y 523.918,Z 267.844,A -85,B 0,C 180,E1 -4719.085,E2 -4719.085} C_VEL
LIN {X 0,Y 523.95,Z 267.843,A -85,B 0,C 180,E1 -4722.119,E2 -4722.119} C_VEL
LIN {X 0,Y 523.94,Z 267.846,A -85,B 0,C 180,E1 -4725.31,E2 -4725.31} C_VEL
LIN {X 0,Y 523.955,Z 267.838,A -85,B 0,C 180,E1 -4728.69,E2 -4728.69} C_VEL
LIN {X 0,Y 523.916,Z 267.847,A -85,B 0,C 180,E1 -4731.081,E2 -4731.081} C_VEL
LIN {X 0,Y 523.923,Z 267.849,A -85,B 0,C 180,E1 -4733.827,E2 -4733.827} C_VEL
LIN {X 0,Y 523.941,Z 267.842,A -85,B 0,C 180,E1 -4736.636,E2 -4736.636} C_VEL
LIN {X 0,Y 523.955,Z 267.846,A -85,B 0,C 180,E1 -4739.356,E2 -4739.356} C_VEL
LIN {X 0,Y 523.961,Z 267.898,A -85,B 0,C 180,E1 -4741.538,E2 -4741.538} C_VEL
LIN {X 0,Y 526.833,Z 280.388,A -85,B 0,C 180,E1 -4743.353,E2 -4743.353} C_VEL
LIN {X 0,Y 526.545,Z 295.403,A -85,B 0,C 180,E1 -4745.304,E2 -4745.304} C_VEL
LIN {X 0,Y 525.862,Z 316.751,A -85,B 0,C 180,E1 -4748.025,E2 -4748.025} C_VEL
LIN {X 0,Y 525.804,Z 320.495,A -85,B 0,C 180,E1 -4748.502,E2 -4748.502} C_VEL
LIN {X 0,Y 528.535,Z 335.663,A -85,B 0,C 180,E1 -4748.837,E2 -4748.837} C_VEL
LIN {X 0,Y 527.538,Z 487.342,A -85,B 0,C 180,E1 -4750.969,E2 -4750.969} C_VEL
LIN {X 0,Y 527.25,Z 502.8,A -85,B 0,C 180,E1 -4751.343,E2 -4751.343} C_VEL
LIN {X 0,Y 526.878,Z 516.939,A -85,B 0,C 180,E1 -4751.833,E2 -4751.833} C_VEL
LIN {X 0,Y 526.469,Z 529.984,A -85,B 0,C 180,E1 -4752.421,E2 -4752.421} C_VEL
LIN {X 0,Y 525.979,Z 543.923,A -85,B 0,C 180,E1 -4753.205,E2 -4753.205} C_VEL
LIN {X 0,Y 525.523,Z 557.219,A -85,B 0,C 180,E1 -4754.129,E2 -4754.129} C_VEL
LIN {X 0,Y 525.031,Z 569.639,A -85,B 0,C 180,E1 -4755.169,E2 -4755.169} C_VEL
LIN {X 0,Y 524.631,Z 580.448,A -85,B 0,C 180,E1 -4756.245,E2 -4756.245} C_VEL
LIN {X 0,Y 524.287,Z 590.468,A -85,B 0,C 180,E1 -4757.419,E2 -4757.419} C_VEL
LIN {X 0,Y 523.983,Z 600.273,A -85,B 0,C 180,E1 -4758.786,E2 -4758.786} C_VEL
LIN {X 0,Y 523.707,Z 608.456,A -85,B 0,C 180,E1 -4760.148,E2 -4760.148} C_VEL
LIN {X 0,Y 523.581,Z 615.223,A -85,B 0,C 180,E1 -4761.509,E2 -4761.509} C_VEL
LIN {X 0,Y 523.48,Z 621.475,A -85,B 0,C 180,E1 -4763.06,E2 -4763.06} C_VEL
LIN {X 0,Y 523.441,Z 626.311,A -85,B 0,C 180,E1 -4764.607,E2 -4764.607} C_VEL
LIN {X 0,Y 523.401,Z 629.854,A -85,B 0,C 180,E1 -4766.151,E2 -4766.151} C_VEL
LIN {X 0,Y 523.332,Z 632.18,A -85,B 0,C 180,E1 -4767.691,E2 -4767.691} C_VEL
LIN {X 0,Y 523.248,Z 633.345,A -85,B 0,C 180,E1 -4769.231,E2 -4769.231} C_VEL
LIN {X 0,Y 523.248,Z 633.344,A -85,B 0,C 180,E1 -4770.77,E2 -4770.77} C_VEL
LIN {X 0,Y 523.332,Z 632.175,A -85,B 0,C 180,E1 -4772.309,E2 -4772.309} C_VEL
LIN {X 0,Y 523.401,Z 629.847,A -85,B 0,C 180,E1 -4773.85,E2 -4773.85} C_VEL
LIN {X 0,Y 523.441,Z 626.31,A -85,B 0,C 180,E1 -4775.393,E2 -4775.393} C_VEL
LIN {X 0,Y 523.481,Z 621.476,A -85,B 0,C 180,E1 -4776.94,E2 -4776.94} C_VEL
LIN {X 0,Y 523.581,Z 615.216,A -85,B 0,C 180,E1 -4778.491,E2 -4778.491} C_VEL
LIN {X 0,Y 523.776,Z 607.357,A -85,B 0,C 180,E1 -4780.046,E2 -4780.046} C_VEL
LIN {X 0,Y 524.014,Z 599,A -85,B 0,C 180,E1 -4781.41,E2 -4781.41} C_VEL
LIN {X 0,Y 524.348,Z 588.937,A -85,B 0,C 180,E1 -4782.777,E2 -4782.777} C_VEL
LIN {X 0,Y 524.707,Z 578.646,A -85,B 0,C 180,E1 -4783.952,E2 -4783.952} C_VEL
LIN {X 0,Y 525.192,Z 566.394,A -85,B 0,C 180,E1 -4785.127,E2 -4785.127} C_VEL
LIN {X 0,Y 525.675,Z 552.761,A -85,B 0,C 180,E1 -4786.206,E2 -4786.206} C_VEL
LIN {X 0,Y 526.215,Z 539.098,A -85,B 0,C 180,E1 -4787.088,E2 -4787.088} C_VEL
LIN {X 0,Y 526.628,Z 524.952,A -85,B 0,C 180,E1 -4787.825,E2 -4787.825} C_VEL
LIN {X 0,Y 527.026,Z 510.403,A -85,B 0,C 180,E1 -4788.414,E2 -4788.414} C_VEL
LIN {X 0,Y 527.387,Z 495.181,A -85,B 0,C 180,E1 -4788.863,E2 -4788.863} C_VEL
LIN {X 0,Y 527.629,Z 479.497,A -85,B 0,C 180,E1 -4789.16,E2 -4789.16} C_VEL
LIN {X 0,Y 528.502,Z 334.622,A -85,B 0,C 180,E1 -4791.179,E2 -4791.179} C_VEL
LIN {X 0,Y 525.785,Z 320.34,A -85,B 0,C 180,E1 -4791.519,E2 -4791.519} C_VEL
LIN {X 0,Y 526.453,Z 297.354,A -85,B 0,C 180,E1 -4794.447,E2 -4794.447} C_VEL
LIN {X 0,Y 526.937,Z 281.511,A -85,B 0,C 180,E1 -4796.494,E2 -4796.494} C_VEL
LIN {X 0,Y 525.588,Z 274.684,A -85,B 0,C 180,E1 -4797.466,E2 -4797.466} C_VEL
LIN {X 0,Y 523.954,Z 267.848,A -85,B 0,C 180,E1 -4798.491,E2 -4798.491} C_VEL
LIN {X 0,Y 523.923,Z 267.845,A -85,B 0,C 180,E1 -4801.545,E2 -4801.545} C_VEL
LIN {X 0,Y 523.935,Z 267.849,A -85,B 0,C 180,E1 -4804.291,E2 -4804.291} C_VEL
LIN {X 0,Y 523.91,Z 267.846,A -85,B 0,C 180,E1 -4807.133,E2 -4807.133} C_VEL
LIN {X 0,Y 523.94,Z 267.842,A -85,B 0,C 180,E1 -4810.13,E2 -4810.13} C_VEL
